REGION Network 3: Дискретные входы состояния НБ
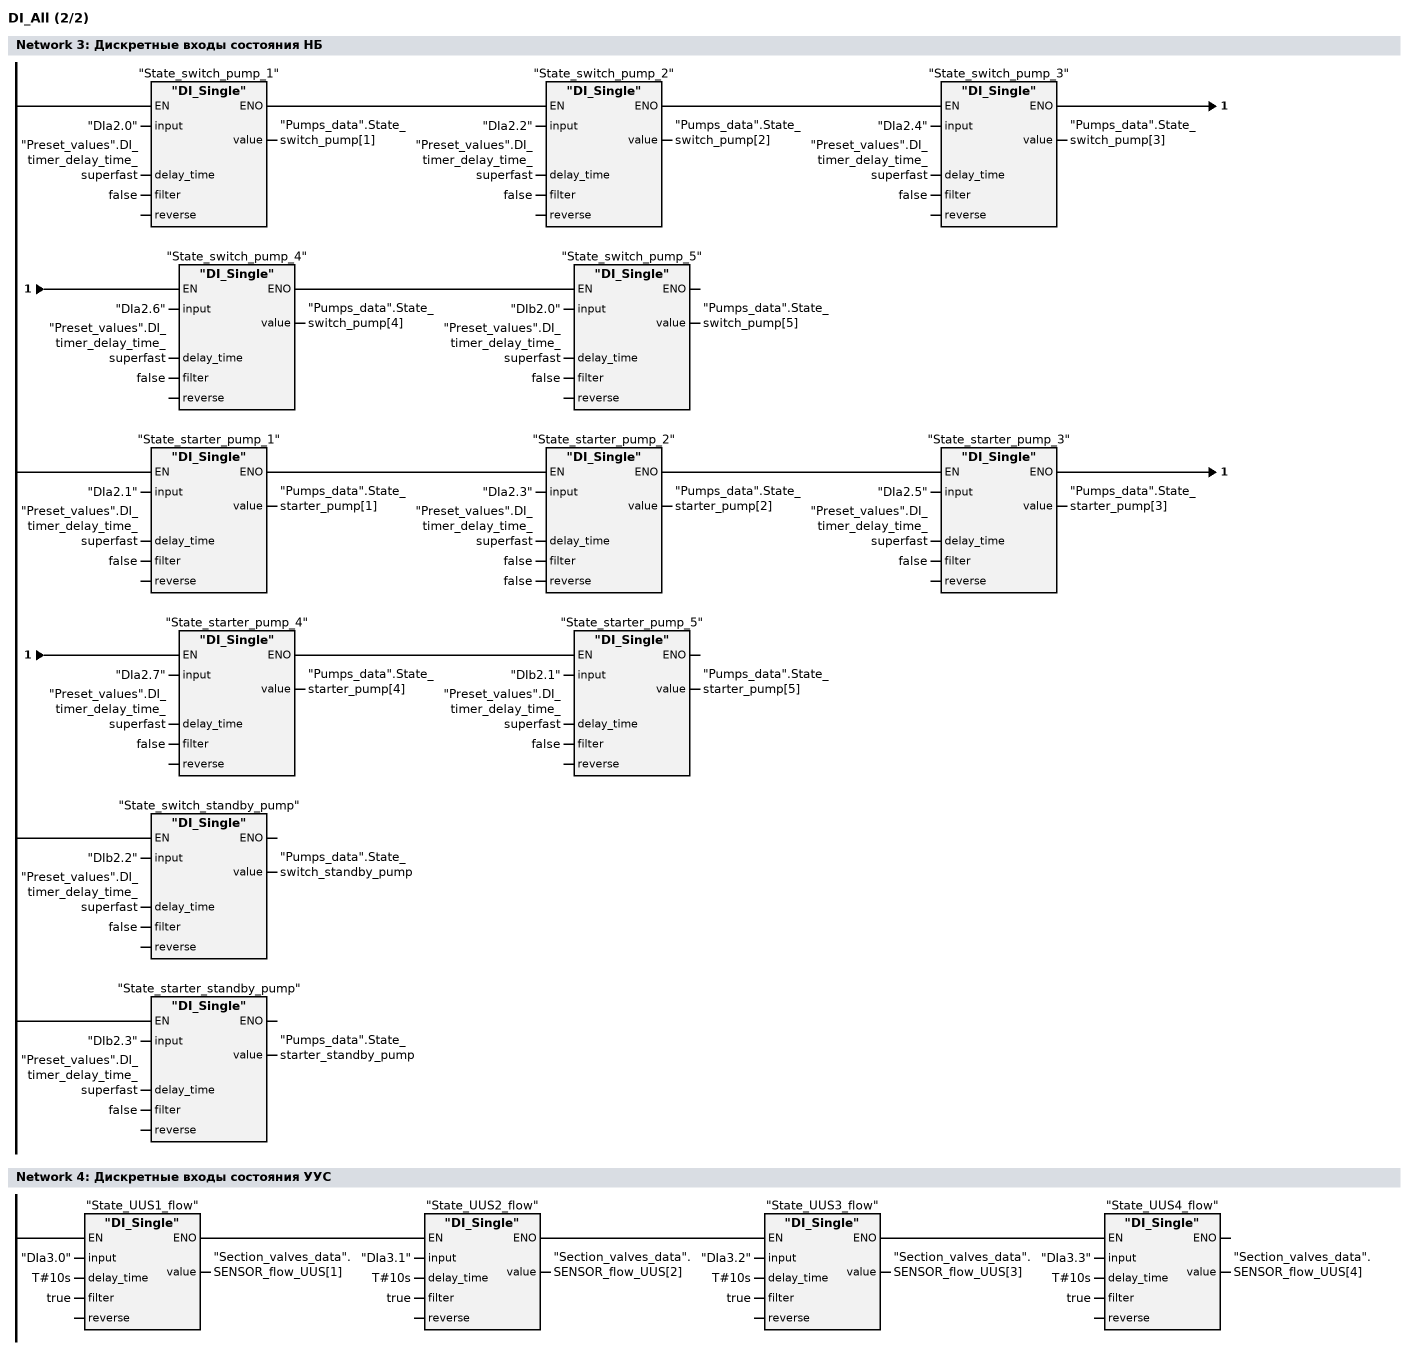
   RUNG wire#powerrail
      "State_switch_pump_1"(input := "DIa2.0", delay_time := "Preset_values".DI_timer_delay_time_superfast, filter := false, reverse :=, value => "Pumps_data".State_switch_pump[1])
      "State_switch_pump_2"(input := "DIa2.2", delay_time := "Preset_values".DI_timer_delay_time_superfast, filter := false, reverse :=, value => "Pumps_data".State_switch_pump[2])
      "State_switch_pump_3"(input := "DIa2.4", delay_time := "Preset_values".DI_timer_delay_time_superfast, filter := false, reverse :=, value => "Pumps_data".State_switch_pump[3])
      "State_switch_pump_4"(input := "DIa2.6", delay_time := "Preset_values".DI_timer_delay_time_superfast, filter := false, reverse :=, value => "Pumps_data".State_switch_pump[4])
      "State_switch_pump_5"(input := "DIb2.0", delay_time := "Preset_values".DI_timer_delay_time_superfast, filter := false, reverse :=, value => "Pumps_data".State_switch_pump[5])
   END_RUNG
   RUNG wire#powerrail
      "State_starter_pump_1"(input := "DIa2.1", delay_time := "Preset_values".DI_timer_delay_time_superfast, filter := false, reverse :=, value => "Pumps_data".State_starter_pump[1])
      "State_starter_pump_2"(input := "DIa2.3", delay_time := "Preset_values".DI_timer_delay_time_superfast, filter := false, reverse := false, value => "Pumps_data".State_starter_pump[2])
      "State_starter_pump_3"(input := "DIa2.5", delay_time := "Preset_values".DI_timer_delay_time_superfast, filter := false, reverse :=, value => "Pumps_data".State_starter_pump[3])
      "State_starter_pump_4"(input := "DIa2.7", delay_time := "Preset_values".DI_timer_delay_time_superfast, filter := false, reverse :=, value => "Pumps_data".State_starter_pump[4])
      "State_starter_pump_5"(input := "DIb2.1", delay_time := "Preset_values".DI_timer_delay_time_superfast, filter := false, reverse :=, value => "Pumps_data".State_starter_pump[5])
   END_RUNG
   RUNG wire#powerrail
      "State_switch_standby_pump"(input := "DIb2.2", delay_time := "Preset_values".DI_timer_delay_time_superfast, filter := false, reverse :=, value => "Pumps_data".State_switch_standby_pump)
   END_RUNG
   RUNG wire#powerrail
      "State_starter_standby_pump"(input := "DIb2.3", delay_time := "Preset_values".DI_timer_delay_time_superfast, filter := false, reverse :=, value => "Pumps_data".State_starter_standby_pump)
   END_RUNG
   // the same network as SCL:
   "State_switch_pump_1"(input := "DIa2.0",   // "DI_Single"
                         delay_time := "Preset_values".DI_timer_delay_time_superfast,
                         filter := false,
                         value => "Pumps_data".State_switch_pump[1],
                         ENO => #_w1);
   "State_switch_pump_2"(EN := #_w1,   // "DI_Single"
                         input := "DIa2.2",
                         delay_time := "Preset_values".DI_timer_delay_time_superfast,
                         filter := false,
                         value => "Pumps_data".State_switch_pump[2],
                         ENO => #_w2);
   "State_switch_pump_3"(EN := #_w2,   // "DI_Single"
                         input := "DIa2.4",
                         delay_time := "Preset_values".DI_timer_delay_time_superfast,
                         filter := false,
                         value => "Pumps_data".State_switch_pump[3],
                         ENO => #_w3);
   "State_switch_pump_4"(EN := #_w3,   // "DI_Single"
                         input := "DIa2.6",
                         delay_time := "Preset_values".DI_timer_delay_time_superfast,
                         filter := false,
                         value => "Pumps_data".State_switch_pump[4],
                         ENO => #_w4);
   IF #_w4 THEN
       "State_switch_pump_5"(input := "DIb2.0",   // "DI_Single"
                             delay_time := "Preset_values".DI_timer_delay_time_superfast,
                             filter := false,
                             value => "Pumps_data".State_switch_pump[5]);
   END_IF;
   "State_starter_pump_1"(input := "DIa2.1",   // "DI_Single"
                          delay_time := "Preset_values".DI_timer_delay_time_superfast,
                          filter := false,
                          value => "Pumps_data".State_starter_pump[1],
                          ENO => #_w5);
   "State_starter_pump_2"(EN := #_w5,   // "DI_Single"
                          input := "DIa2.3",
                          delay_time := "Preset_values".DI_timer_delay_time_superfast,
                          filter := false,
                          reverse := false,
                          value => "Pumps_data".State_starter_pump[2],
                          ENO => #_w6);
   "State_starter_pump_3"(EN := #_w6,   // "DI_Single"
                          input := "DIa2.5",
                          delay_time := "Preset_values".DI_timer_delay_time_superfast,
                          filter := false,
                          value => "Pumps_data".State_starter_pump[3],
                          ENO => #_w7);
   "State_starter_pump_4"(EN := #_w7,   // "DI_Single"
                          input := "DIa2.7",
                          delay_time := "Preset_values".DI_timer_delay_time_superfast,
                          filter := false,
                          value => "Pumps_data".State_starter_pump[4],
                          ENO => #_w8);
   IF #_w8 THEN
       "State_starter_pump_5"(input := "DIb2.1",   // "DI_Single"
                              delay_time := "Preset_values".DI_timer_delay_time_superfast,
                              filter := false,
                              value => "Pumps_data".State_starter_pump[5]);
   END_IF;
   "State_switch_standby_pump"(input := "DIb2.2",   // "DI_Single"
                           delay_time := "Preset_values".DI_timer_delay_time_superfast,
                           filter := false,
                           value => "Pumps_data".State_switch_standby_pump);
   "State_starter_standby_pump"(input := "DIb2.3",   // "DI_Single"
                           delay_time := "Preset_values".DI_timer_delay_time_superfast,
                           filter := false,
                           value => "Pumps_data".State_starter_standby_pump);
END_REGION

REGION Network 4: Дискретные входы состояния УУС
   RUNG wire#powerrail
      "State_UUS1_flow"(input := "DIa3.0", delay_time := T#10s, filter := true, reverse :=, value => "Section_valves_data".SENSOR_flow_UUS[1])
      "State_UUS2_flow"(input := "DIa3.1", delay_time := T#10s, filter := true, reverse :=, value => "Section_valves_data".SENSOR_flow_UUS[2])
      "State_UUS3_flow"(input := "DIa3.2", delay_time := T#10s, filter := true, reverse :=, value => "Section_valves_data".SENSOR_flow_UUS[3])
      "State_UUS4_flow"(input := "DIa3.3", delay_time := T#10s, filter := true, reverse :=, value => "Section_valves_data".SENSOR_flow_UUS[4])
   END_RUNG
   // the same network as SCL:
   "State_UUS1_flow"(input := "DIa3.0",   // "DI_Single"
                     delay_time := T#10s,
                     filter := true,
                     value => "Section_valves_data".SENSOR_flow_UUS[1],
                     ENO => #_w1);
   "State_UUS2_flow"(EN := #_w1,   // "DI_Single"
                     input := "DIa3.1",
                     delay_time := T#10s,
                     filter := true,
                     value => "Section_valves_data".SENSOR_flow_UUS[2],
                     ENO => #_w2);
   "State_UUS3_flow"(EN := #_w2,   // "DI_Single"
                     input := "DIa3.2",
                     delay_time := T#10s,
                     filter := true,
                     value => "Section_valves_data".SENSOR_flow_UUS[3],
                     ENO => #_w3);
   IF #_w3 THEN
       "State_UUS4_flow"(input := "DIa3.3",   // "DI_Single"
                         delay_time := T#10s,
                         filter := true,
                         value => "Section_valves_data".SENSOR_flow_UUS[4]);
   END_IF;
END_REGION
END_FUNCTION

FUNCTION "AI_All" : Void   // FC2, LAD
{ S7_Optimized_Access := 'TRUE' }
VERSION : 0.1
   VAR_TEMP   // added for the SCL form of the ladder/FBD networks
      _w1 : Bool;
      _w2 : Bool;
      _w3 : Bool;
      _w4 : Bool;
   END_VAR
BEGIN

REGION Network 1: Аналоговые входы датчиков низкого давления
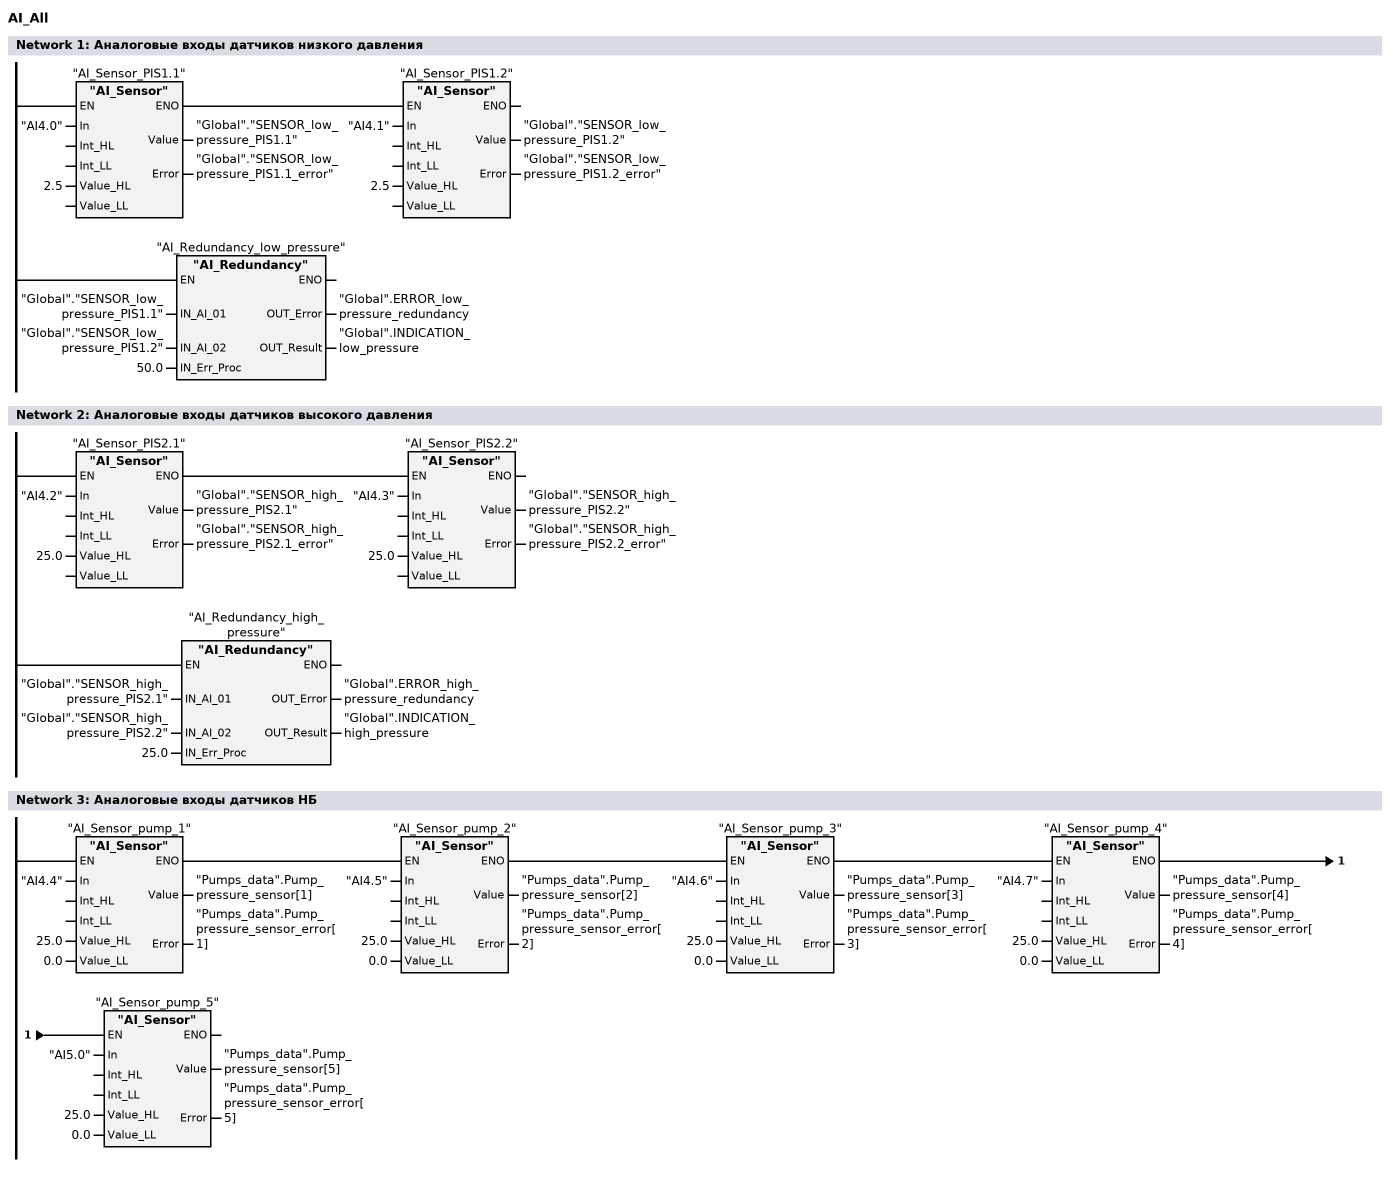
   RUNG wire#powerrail
      "AI_Sensor_PIS1.1"(In := "AI4.0", Int_HL :=, Int_LL :=, Value_HL := 2.5, Value_LL :=, Value => "Global"."SENSOR_low_pressure_PIS1.1", Error => "Global"."SENSOR_low_pressure_PIS1.1_error")
      "AI_Sensor_PIS1.2"(In := "AI4.1", Int_HL :=, Int_LL :=, Value_HL := 2.5, Value_LL :=, Value => "Global"."SENSOR_low_pressure_PIS1.2", Error => "Global"."SENSOR_low_pressure_PIS1.2_error")
   END_RUNG
   RUNG wire#powerrail
      "AI_Redundancy_low_pressure"(IN_AI_01 := "Global"."SENSOR_low_pressure_PIS1.1", IN_AI_02 := "Global"."SENSOR_low_pressure_PIS1.2", IN_Err_Proc := 50.0, OUT_Error => "Global".ERROR_low_pressure_redundancy, OUT_Result => "Global".INDICATION_low_pressure)
   END_RUNG
   // the same network as SCL:
   "AI_Sensor_PIS1.1"(In := "AI4.0",   // "AI_Sensor"
                      Value_HL := 2.5,
                      Value => "Global"."SENSOR_low_pressure_PIS1.1",
                      Error => "Global"."SENSOR_low_pressure_PIS1.1_error",
                      ENO => #_w1);
   IF #_w1 THEN
       "AI_Sensor_PIS1.2"(In := "AI4.1",   // "AI_Sensor"
                          Value_HL := 2.5,
                          Value => "Global"."SENSOR_low_pressure_PIS1.2",
                          Error => "Global"."SENSOR_low_pressure_PIS1.2_error");
   END_IF;
   "AI_Redundancy_low_pressure"(IN_AI_01 := "Global"."SENSOR_low_pressure_PIS1.1",   // "AI_Redundancy"
                           IN_AI_02 := "Global"."SENSOR_low_pressure_PIS1.2",
                           IN_Err_Proc := 50.0,
                           OUT_Error => "Global".ERROR_low_pressure_redundancy,
                           OUT_Result => "Global".INDICATION_low_pressure);
END_REGION

REGION Network 2: Аналоговые входы датчиков высокого давления
   RUNG wire#powerrail
      "AI_Sensor_PIS2.1"(In := "AI4.2", Int_HL :=, Int_LL :=, Value_HL := 25.0, Value_LL :=, Value => "Global"."SENSOR_high_pressure_PIS2.1", Error => "Global"."SENSOR_high_pressure_PIS2.1_error")
      "AI_Sensor_PIS2.2"(In := "AI4.3", Int_HL :=, Int_LL :=, Value_HL := 25.0, Value_LL :=, Value => "Global"."SENSOR_high_pressure_PIS2.2", Error => "Global"."SENSOR_high_pressure_PIS2.2_error")
   END_RUNG
   RUNG wire#powerrail
      "AI_Redundancy_high_pressure"(IN_AI_01 := "Global"."SENSOR_high_pressure_PIS2.1", IN_AI_02 := "Global"."SENSOR_high_pressure_PIS2.2", IN_Err_Proc := 25.0, OUT_Error => "Global".ERROR_high_pressure_redundancy, OUT_Result => "Global".INDICATION_high_pressure)
   END_RUNG
   // the same network as SCL:
   "AI_Sensor_PIS2.1"(In := "AI4.2",   // "AI_Sensor"
                      Value_HL := 25.0,
                      Value => "Global"."SENSOR_high_pressure_PIS2.1",
                      Error => "Global"."SENSOR_high_pressure_PIS2.1_error",
                      ENO => #_w1);
   IF #_w1 THEN
       "AI_Sensor_PIS2.2"(In := "AI4.3",   // "AI_Sensor"
                          Value_HL := 25.0,
                          Value => "Global"."SENSOR_high_pressure_PIS2.2",
                          Error => "Global"."SENSOR_high_pressure_PIS2.2_error");
   END_IF;
   "AI_Redundancy_high_pressure"(IN_AI_01 := "Global"."SENSOR_high_pressure_PIS2.1",   // "AI_Redundancy"
                           IN_AI_02 := "Global"."SENSOR_high_pressure_PIS2.2",
                           IN_Err_Proc := 25.0,
                           OUT_Error => "Global".ERROR_high_pressure_redundancy,
                           OUT_Result => "Global".INDICATION_high_pressure);
END_REGION

REGION Network 3: Аналоговые входы датчиков НБ
   RUNG wire#powerrail
      "AI_Sensor_pump_1"(In := "AI4.4", Int_HL :=, Int_LL :=, Value_HL := 25.0, Value_LL := 0.0, Value => "Pumps_data".Pump_pressure_sensor[1], Error => "Pumps_data".Pump_pressure_sensor_error[1])
      "AI_Sensor_pump_2"(In := "AI4.5", Int_HL :=, Int_LL :=, Value_HL := 25.0, Value_LL := 0.0, Value => "Pumps_data".Pump_pressure_sensor[2], Error => "Pumps_data".Pump_pressure_sensor_error[2])
      "AI_Sensor_pump_3"(In := "AI4.6", Int_HL :=, Int_LL :=, Value_HL := 25.0, Value_LL := 0.0, Value => "Pumps_data".Pump_pressure_sensor[3], Error => "Pumps_data".Pump_pressure_sensor_error[3])
      "AI_Sensor_pump_4"(In := "AI4.7", Int_HL :=, Int_LL :=, Value_HL := 25.0, Value_LL := 0.0, Value => "Pumps_data".Pump_pressure_sensor[4], Error => "Pumps_data".Pump_pressure_sensor_error[4])
      "AI_Sensor_pump_5"(In := "AI5.0", Int_HL :=, Int_LL :=, Value_HL := 25.0, Value_LL := 0.0, Value => "Pumps_data".Pump_pressure_sensor[5], Error => "Pumps_data".Pump_pressure_sensor_error[5])
   END_RUNG
   // the same network as SCL:
   "AI_Sensor_pump_1"(In := "AI4.4",   // "AI_Sensor"
                      Value_HL := 25.0,
                      Value_LL := 0.0,
                      Value => "Pumps_data".Pump_pressure_sensor[1],
                      Error => "Pumps_data".Pump_pressure_sensor_error[1],
                      ENO => #_w1);
   "AI_Sensor_pump_2"(EN := #_w1,   // "AI_Sensor"
                      In := "AI4.5",
                      Value_HL := 25.0,
                      Value_LL := 0.0,
                      Value => "Pumps_data".Pump_pressure_sensor[2],
                      Error => "Pumps_data".Pump_pressure_sensor_error[2],
                      ENO => #_w2);
   "AI_Sensor_pump_3"(EN := #_w2,   // "AI_Sensor"
                      In := "AI4.6",
                      Value_HL := 25.0,
                      Value_LL := 0.0,
                      Value => "Pumps_data".Pump_pressure_sensor[3],
                      Error => "Pumps_data".Pump_pressure_sensor_error[3],
                      ENO => #_w3);
   "AI_Sensor_pump_4"(EN := #_w3,   // "AI_Sensor"
                      In := "AI4.7",
                      Value_HL := 25.0,
                      Value_LL := 0.0,
                      Value => "Pumps_data".Pump_pressure_sensor[4],
                      Error => "Pumps_data".Pump_pressure_sensor_error[4],
                      ENO => #_w4);
   IF #_w4 THEN
       "AI_Sensor_pump_5"(In := "AI5.0",   // "AI_Sensor"
                          Value_HL := 25.0,
                          Value_LL := 0.0,
                          Value => "Pumps_data".Pump_pressure_sensor[5],
                          Error => "Pumps_data".Pump_pressure_sensor_error[5]);
   END_IF;
END_REGION
END_FUNCTION

ORGANIZATION_BLOCK "Main"   // OB1, LAD, ProgramCycle
TITLE = "Main Program Sweep (Cycle)"
{ S7_Optimized_Access := 'TRUE' }
VERSION : 0.1
   VAR_INPUT
      Initial_Call : Bool;   // Initial call of this OB
      Remanence : Bool;   // =True, if remanent data are available
   END_VAR
BEGIN

REGION Network 1: Обработка дискретных и аналоговых сигналов
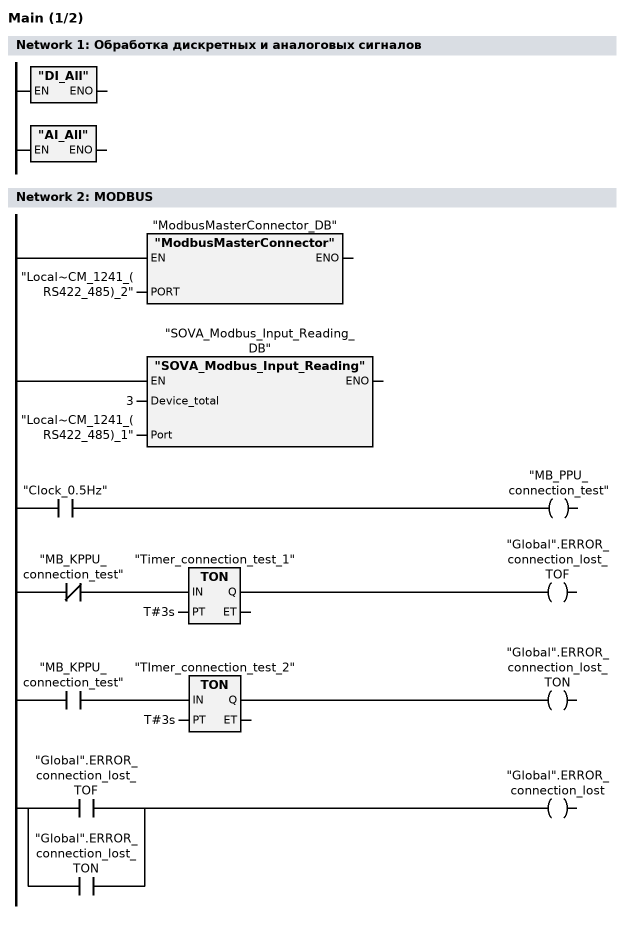
   RUNG wire#powerrail
      "DI_All"()
   END_RUNG
   RUNG wire#powerrail
      "AI_All"()
   END_RUNG
   // the same network as SCL:
   "DI_All"();
   "AI_All"();
END_REGION

REGION Network 2: MODBUS
   "ModbusMasterConnector_DB"(PORT := "Local~CM_1241_(RS422_485)_2");   // "ModbusMasterConnector"
   "SOVA_Modbus_Input_Reading_DB"(Device_total := 3, Port := "Local~CM_1241_(RS422_485)_1");   // "SOVA_Modbus_Input_Reading"
   "MB_PPU_connection_test" := "Clock_0.5Hz";
   "Timer_connection_test_1".TON(IN := NOT "MB_KPPU_connection_test", PT := T#3s);
   "Global".ERROR_connection_lost_TOF := "Timer_connection_test_1".Q;
   "TImer_connection_test_2".TON(IN := "MB_KPPU_connection_test", PT := T#3s);
   "Global".ERROR_connection_lost_TON := "TImer_connection_test_2".Q;
   "Global".ERROR_connection_lost := "Global".ERROR_connection_lost_TOF OR "Global".ERROR_connection_lost_TON;
END_REGION

REGION Network 3: Состояние режима работы ППУ
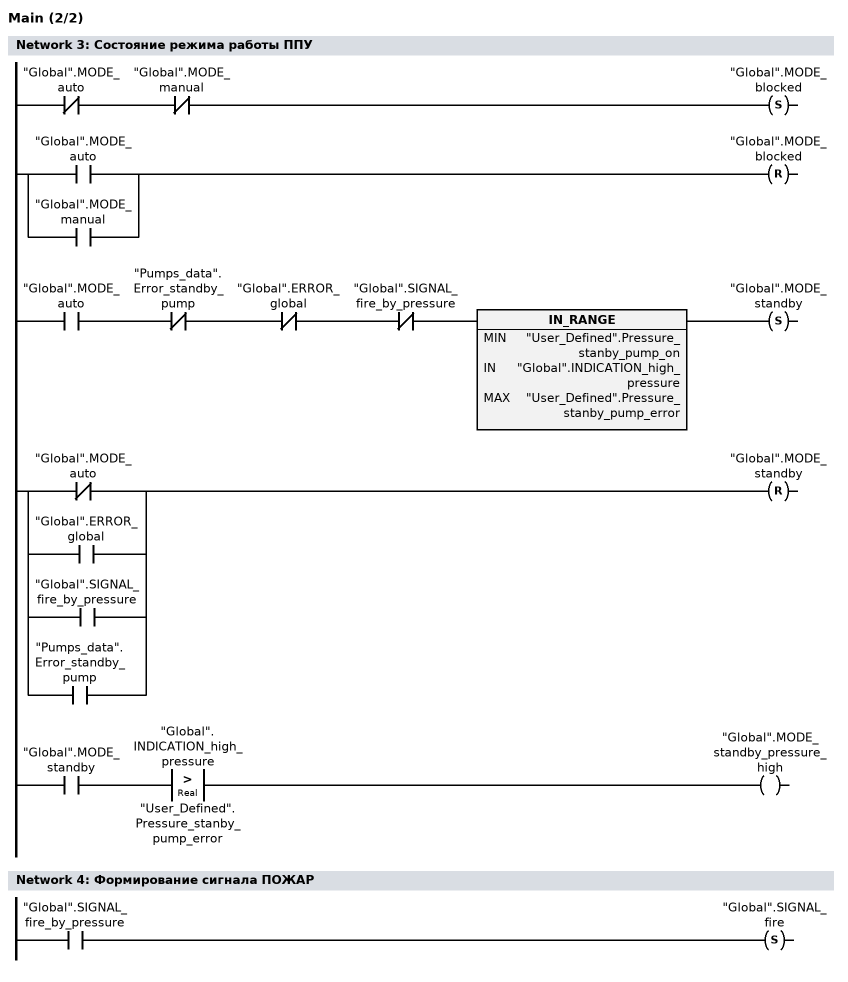
   RUNG wire#powerrail
      I_Contact( "Global".MODE_auto )
      I_Contact( "Global".MODE_manual )
      S_Coil( "Global".MODE_blocked )
   END_RUNG
   RUNG wire#powerrail
      Contact( "Global".MODE_auto )
      wire#w1
      R_Coil( "Global".MODE_blocked )
   END_RUNG
   RUNG wire#powerrail
      Contact( "Global".MODE_manual )
   END_RUNG wire#w1
   RUNG wire#powerrail
      Contact( "Global".MODE_auto )
      I_Contact( "Pumps_data".Error_standby_pump )
      I_Contact( "Global".ERROR_global )
      I_Contact( "Global".SIGNAL_fire_by_pressure )
      { S7_Templates := "SrcType := Real" } InRange(min := "User_Defined".Pressure_stanby_pump_on, in := "Global".INDICATION_high_pressure, max := "User_Defined".Pressure_stanby_pump_error)
      S_Coil( "Global".MODE_standby )
   END_RUNG
   RUNG wire#powerrail
      I_Contact( "Global".MODE_auto )
      wire#w2
      R_Coil( "Global".MODE_standby )
   END_RUNG
   RUNG wire#powerrail
      Contact( "Global".ERROR_global )
   END_RUNG wire#w2
   RUNG wire#powerrail
      Contact( "Global".SIGNAL_fire_by_pressure )
   END_RUNG wire#w2
   RUNG wire#powerrail
      Contact( "Pumps_data".Error_standby_pump )
   END_RUNG wire#w2
   RUNG wire#powerrail
      Contact( "Global".MODE_standby )
      { S7_Templates := "SrcType := Real" } GT_Contact(in1 := "Global".INDICATION_high_pressure, in2 := "User_Defined".Pressure_stanby_pump_error)
      Coil( "Global".MODE_standby_pressure_high )
   END_RUNG
   // the same network as SCL:
   IF NOT "Global".MODE_auto AND NOT "Global".MODE_manual THEN "Global".MODE_blocked := TRUE; END_IF;
   IF "Global".MODE_auto OR "Global".MODE_manual THEN "Global".MODE_blocked := FALSE; END_IF;
   IF "Global".MODE_auto AND NOT "Pumps_data".Error_standby_pump AND NOT "Global".ERROR_global AND NOT "Global".SIGNAL_fire_by_pressure AND ("User_Defined".Pressure_stanby_pump_on <= "Global".INDICATION_high_pressure) AND ("Global".INDICATION_high_pressure <= "User_Defined".Pressure_stanby_pump_error) THEN
       "Global".MODE_standby := TRUE;
   END_IF;
   IF NOT "Global".MODE_auto OR "Global".ERROR_global OR "Global".SIGNAL_fire_by_pressure OR "Pumps_data".Error_standby_pump THEN
       "Global".MODE_standby := FALSE;
   END_IF;
   "Global".MODE_standby_pressure_high := "Global".MODE_standby AND ("Global".INDICATION_high_pressure > "User_Defined".Pressure_stanby_pump_error);
END_REGION

REGION Network 4: Формирование сигнала ПОЖАР
   RUNG wire#powerrail
      Contact( "Global".SIGNAL_fire_by_pressure )
      S_Coil( "Global".SIGNAL_fire )
   END_RUNG
   // the same network as SCL:
   IF "Global".SIGNAL_fire_by_pressure THEN "Global".SIGNAL_fire := TRUE; END_IF;
END_REGION

REGION Network 5 (SCL): Pump Work Counter
   IF "Pumps_data".State_work_pump[1] THEN
       "Pumps_data".Pump_work_counter_arr[1] := 1;
   ELSE
       "Pumps_data".Pump_work_counter_arr[1] := 0;
   END_IF;

   IF "Pumps_data".State_work_pump[2] THEN
       "Pumps_data".Pump_work_counter_arr[2] := 1;
   ELSE
       "Pumps_data".Pump_work_counter_arr[2] := 0;
   END_IF;

   IF "Pumps_data".State_work_pump[3] THEN
       "Pumps_data".Pump_work_counter_arr[3] := 1;
   ELSE
       "Pumps_data".Pump_work_counter_arr[3] := 0;
   END_IF;

   IF "Pumps_data".State_work_pump[4] THEN
       "Pumps_data".Pump_work_counter_arr[4] := 1;
   ELSE
       "Pumps_data".Pump_work_counter_arr[4] := 0;
   END_IF;

   IF "Pumps_data".State_work_pump[5] THEN
       "Pumps_data".Pump_work_counter_arr[5] := 1;
   ELSE
       "Pumps_data".Pump_work_counter_arr[5] := 0;
   END_IF;

   IF "Pumps_data".State_work_pump[6] THEN
       "Pumps_data".Pump_work_counter_arr[6] := 1;
   ELSE
       "Pumps_data".Pump_work_counter_arr[6] := 0;
   END_IF;

   IF "Pumps_data".State_work_pump[7] THEN
       "Pumps_data".Pump_work_counter_arr[7] := 1;
   ELSE
       "Pumps_data".Pump_work_counter_arr[7] := 0;
   END_IF;

   IF "Pumps_data".State_work_pump[8] THEN
       "Pumps_data".Pump_work_counter_arr[8] := 1;
   ELSE
       "Pumps_data".Pump_work_counter_arr[8] := 0;
   END_IF;

   IF "Pumps_data".State_work_pump[9] THEN
       "Pumps_data".Pump_work_counter_arr[9] := 1;
   ELSE
       "Pumps_data".Pump_work_counter_arr[9] := 0;
   END_IF;

   IF "Pumps_data".State_work_pump[10] THEN
       "Pumps_data".Pump_work_counter_arr[10] := 1;
   ELSE
       "Pumps_data".Pump_work_counter_arr[10] := 0;
   END_IF;

   "Pumps_data".pump_work_counter := "Pumps_data".Pump_work_counter_arr[1] +
   "Pumps_data".Pump_work_counter_arr[2] + "Pumps_data".Pump_work_counter_arr[3] +
   "Pumps_data".Pump_work_counter_arr[4] + "Pumps_data".Pump_work_counter_arr[5] +
   "Pumps_data".Pump_work_counter_arr[6] + "Pumps_data".Pump_work_counter_arr[7] +
   "Pumps_data".Pump_work_counter_arr[8] + "Pumps_data".Pump_work_counter_arr[9] +
   "Pumps_data".Pump_work_counter_arr[10];
END_REGION
END_ORGANIZATION_BLOCK

ORGANIZATION_BLOCK "Errors"   // OB123, LAD, ProgramCycle
TITLE = "Main Program Sweep (Cycle)"
{ S7_Optimized_Access := 'TRUE' }
VERSION : 0.1
   VAR_INPUT
      Initial_Call : Bool;   // Initial call of this OB
      Remanence : Bool;   // =True, if remanent data are available
   END_VAR
   VAR_TEMP   // added for the SCL form of the ladder/FBD networks
      _w1 : Bool;
      _w2 : Bool;
      _w3 : Bool;
      _w4 : Bool;
      _w5 : Bool;
      _w6 : Bool;
      _w7 : Bool;
      _w8 : Bool;
   END_VAR
BEGIN

REGION Network 1: Недостаточное входное давление
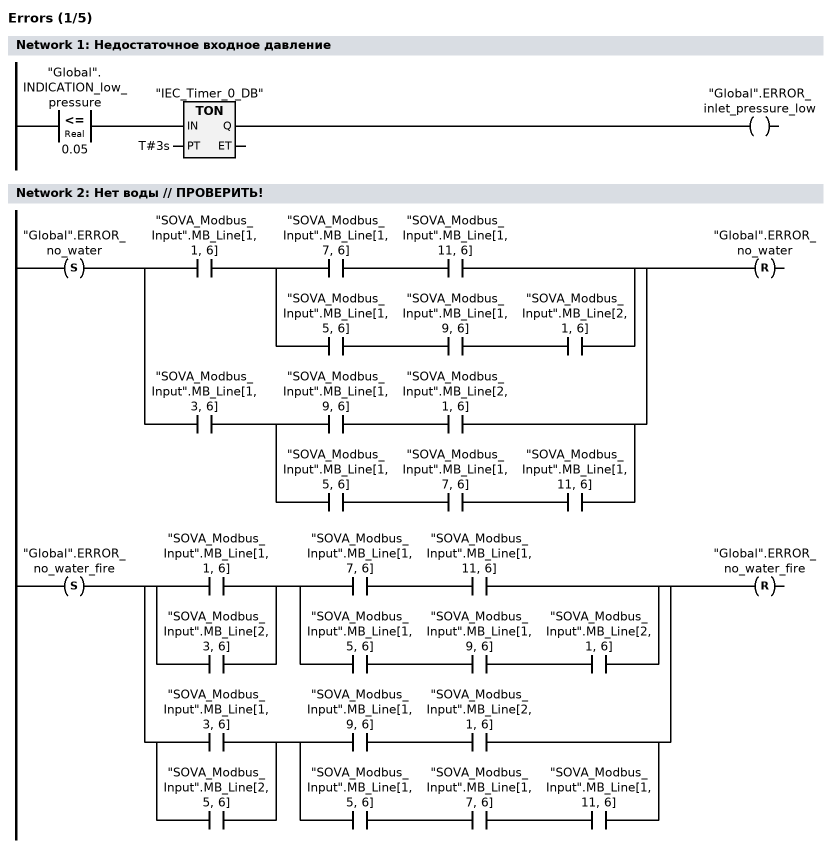
   "IEC_Timer_0_DB".TON(IN := "Global".INDICATION_low_pressure <= 0.05, PT := T#3s);
   "Global".ERROR_inlet_pressure_low := "IEC_Timer_0_DB".Q;
END_REGION

REGION Network 2: Нет воды // ПРОВЕРИТЬ!
   RUNG wire#powerrail
      S_Coil( "Global".ERROR_no_water )
      wire#w1
      Contact( "SOVA_Modbus_Input".MB_Line[1, 1, 6] )
      wire#w2
      Contact( "SOVA_Modbus_Input".MB_Line[1, 7, 6] )
      Contact( "SOVA_Modbus_Input".MB_Line[1, 11, 6] )
      wire#w3
      R_Coil( "Global".ERROR_no_water )
   END_RUNG
   RUNG wire#w2
      Contact( "SOVA_Modbus_Input".MB_Line[1, 5, 6] )
      Contact( "SOVA_Modbus_Input".MB_Line[1, 9, 6] )
      Contact( "SOVA_Modbus_Input".MB_Line[2, 1, 6] )
   END_RUNG wire#w3
   RUNG wire#w1
      Contact( "SOVA_Modbus_Input".MB_Line[1, 3, 6] )
      wire#w4
      Contact( "SOVA_Modbus_Input".MB_Line[1, 9, 6] )
      Contact( "SOVA_Modbus_Input".MB_Line[2, 1, 6] )
   END_RUNG wire#w3
   RUNG wire#w4
      Contact( "SOVA_Modbus_Input".MB_Line[1, 5, 6] )
      Contact( "SOVA_Modbus_Input".MB_Line[1, 7, 6] )
      Contact( "SOVA_Modbus_Input".MB_Line[1, 11, 6] )
   END_RUNG wire#w3
   RUNG wire#powerrail
      S_Coil( "Global".ERROR_no_water_fire )
      wire#w5
      Contact( "SOVA_Modbus_Input".MB_Line[1, 1, 6] )
      wire#w6
      Contact( "SOVA_Modbus_Input".MB_Line[1, 7, 6] )
      Contact( "SOVA_Modbus_Input".MB_Line[1, 11, 6] )
      wire#w7
      R_Coil( "Global".ERROR_no_water_fire )
   END_RUNG
   RUNG wire#w5
      Contact( "SOVA_Modbus_Input".MB_Line[2, 3, 6] )
   END_RUNG wire#w6
   RUNG wire#w6
      Contact( "SOVA_Modbus_Input".MB_Line[1, 5, 6] )
      Contact( "SOVA_Modbus_Input".MB_Line[1, 9, 6] )
      Contact( "SOVA_Modbus_Input".MB_Line[2, 1, 6] )
   END_RUNG wire#w7
   RUNG wire#w5
      Contact( "SOVA_Modbus_Input".MB_Line[1, 3, 6] )
      wire#w8
      Contact( "SOVA_Modbus_Input".MB_Line[1, 9, 6] )
      Contact( "SOVA_Modbus_Input".MB_Line[2, 1, 6] )
   END_RUNG wire#w7
   RUNG wire#w5
      Contact( "SOVA_Modbus_Input".MB_Line[2, 5, 6] )
   END_RUNG wire#w8
   RUNG wire#w8
      Contact( "SOVA_Modbus_Input".MB_Line[1, 5, 6] )
      Contact( "SOVA_Modbus_Input".MB_Line[1, 7, 6] )
      Contact( "SOVA_Modbus_Input".MB_Line[1, 11, 6] )
   END_RUNG wire#w7
   // the same network as SCL:
   "Global".ERROR_no_water := TRUE;
   IF ("SOVA_Modbus_Input".MB_Line[1, 1, 6] AND (("SOVA_Modbus_Input".MB_Line[1, 7, 6] AND "SOVA_Modbus_Input".MB_Line[1, 11, 6]) OR ("SOVA_Modbus_Input".MB_Line[1, 5, 6] AND "SOVA_Modbus_Input".MB_Line[1, 9, 6] AND "SOVA_Modbus_Input".MB_Line[2, 1, 6]))) OR ("SOVA_Modbus_Input".MB_Line[1, 3, 6] AND (("SOVA_Modbus_Input".MB_Line[1, 9, 6] AND "SOVA_Modbus_Input".MB_Line[2, 1, 6]) OR ("SOVA_Modbus_Input".MB_Line[1, 5, 6] AND "SOVA_Modbus_Input".MB_Line[1, 7, 6] AND "SOVA_Modbus_Input".MB_Line[1, 11, 6]))) THEN
       "Global".ERROR_no_water := FALSE;
   END_IF;
   "Global".ERROR_no_water_fire := TRUE;
   IF (("SOVA_Modbus_Input".MB_Line[1, 1, 6] OR "SOVA_Modbus_Input".MB_Line[2, 3, 6]) AND (("SOVA_Modbus_Input".MB_Line[1, 7, 6] AND "SOVA_Modbus_Input".MB_Line[1, 11, 6]) OR ("SOVA_Modbus_Input".MB_Line[1, 5, 6] AND "SOVA_Modbus_Input".MB_Line[1, 9, 6] AND "SOVA_Modbus_Input".MB_Line[2, 1, 6]))) OR (("SOVA_Modbus_Input".MB_Line[1, 3, 6] OR "SOVA_Modbus_Input".MB_Line[2, 5, 6]) AND (("SOVA_Modbus_Input".MB_Line[1, 9, 6] AND "SOVA_Modbus_Input".MB_Line[2, 1, 6]) OR ("SOVA_Modbus_Input".MB_Line[1, 5, 6] AND "SOVA_Modbus_Input".MB_Line[1, 7, 6] AND "SOVA_Modbus_Input".MB_Line[1, 11, 6]))) THEN
       "Global".ERROR_no_water_fire := FALSE;
   END_IF;
END_REGION

REGION Network 3: Неисправность вводных задвижек
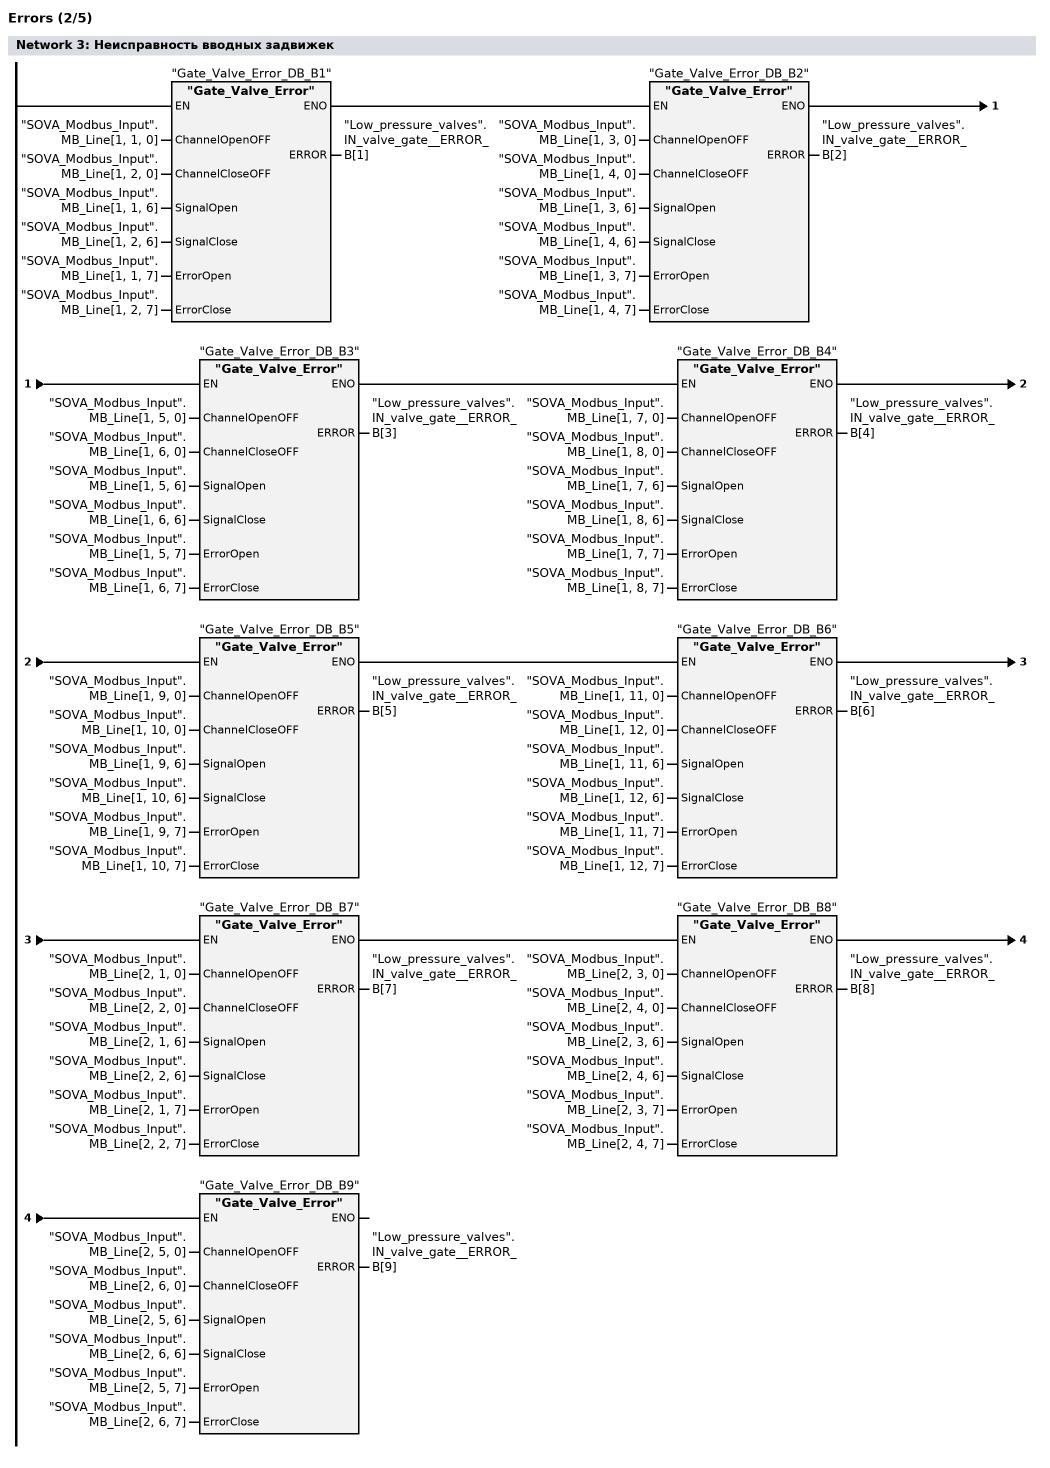
   RUNG wire#powerrail
      "Gate_Valve_Error_DB_B1"(ChannelOpenOFF := "SOVA_Modbus_Input".MB_Line[1, 1, 0], ChannelCloseOFF := "SOVA_Modbus_Input".MB_Line[1, 2, 0], SignalOpen := "SOVA_Modbus_Input".MB_Line[1, 1, 6], SignalClose := "SOVA_Modbus_Input".MB_Line[1, 2, 6], ErrorOpen := "SOVA_Modbus_Input".MB_Line[1, 1, 7], ErrorClose := "SOVA_Modbus_Input".MB_Line[1, 2, 7], ERROR => "Low_pressure_valves".IN_valve_gate__ERROR_B[1])
      "Gate_Valve_Error_DB_B2"(ChannelOpenOFF := "SOVA_Modbus_Input".MB_Line[1, 3, 0], ChannelCloseOFF := "SOVA_Modbus_Input".MB_Line[1, 4, 0], SignalOpen := "SOVA_Modbus_Input".MB_Line[1, 3, 6], SignalClose := "SOVA_Modbus_Input".MB_Line[1, 4, 6], ErrorOpen := "SOVA_Modbus_Input".MB_Line[1, 3, 7], ErrorClose := "SOVA_Modbus_Input".MB_Line[1, 4, 7], ERROR => "Low_pressure_valves".IN_valve_gate__ERROR_B[2])
      "Gate_Valve_Error_DB_B3"(ChannelOpenOFF := "SOVA_Modbus_Input".MB_Line[1, 5, 0], ChannelCloseOFF := "SOVA_Modbus_Input".MB_Line[1, 6, 0], SignalOpen := "SOVA_Modbus_Input".MB_Line[1, 5, 6], SignalClose := "SOVA_Modbus_Input".MB_Line[1, 6, 6], ErrorOpen := "SOVA_Modbus_Input".MB_Line[1, 5, 7], ErrorClose := "SOVA_Modbus_Input".MB_Line[1, 6, 7], ERROR => "Low_pressure_valves".IN_valve_gate__ERROR_B[3])
      "Gate_Valve_Error_DB_B4"(ChannelOpenOFF := "SOVA_Modbus_Input".MB_Line[1, 7, 0], ChannelCloseOFF := "SOVA_Modbus_Input".MB_Line[1, 8, 0], SignalOpen := "SOVA_Modbus_Input".MB_Line[1, 7, 6], SignalClose := "SOVA_Modbus_Input".MB_Line[1, 8, 6], ErrorOpen := "SOVA_Modbus_Input".MB_Line[1, 7, 7], ErrorClose := "SOVA_Modbus_Input".MB_Line[1, 8, 7], ERROR => "Low_pressure_valves".IN_valve_gate__ERROR_B[4])
      "Gate_Valve_Error_DB_B5"(ChannelOpenOFF := "SOVA_Modbus_Input".MB_Line[1, 9, 0], ChannelCloseOFF := "SOVA_Modbus_Input".MB_Line[1, 10, 0], SignalOpen := "SOVA_Modbus_Input".MB_Line[1, 9, 6], SignalClose := "SOVA_Modbus_Input".MB_Line[1, 10, 6], ErrorOpen := "SOVA_Modbus_Input".MB_Line[1, 9, 7], ErrorClose := "SOVA_Modbus_Input".MB_Line[1, 10, 7], ERROR => "Low_pressure_valves".IN_valve_gate__ERROR_B[5])
      "Gate_Valve_Error_DB_B6"(ChannelOpenOFF := "SOVA_Modbus_Input".MB_Line[1, 11, 0], ChannelCloseOFF := "SOVA_Modbus_Input".MB_Line[1, 12, 0], SignalOpen := "SOVA_Modbus_Input".MB_Line[1, 11, 6], SignalClose := "SOVA_Modbus_Input".MB_Line[1, 12, 6], ErrorOpen := "SOVA_Modbus_Input".MB_Line[1, 11, 7], ErrorClose := "SOVA_Modbus_Input".MB_Line[1, 12, 7], ERROR => "Low_pressure_valves".IN_valve_gate__ERROR_B[6])
      "Gate_Valve_Error_DB_B7"(ChannelOpenOFF := "SOVA_Modbus_Input".MB_Line[2, 1, 0], ChannelCloseOFF := "SOVA_Modbus_Input".MB_Line[2, 2, 0], SignalOpen := "SOVA_Modbus_Input".MB_Line[2, 1, 6], SignalClose := "SOVA_Modbus_Input".MB_Line[2, 2, 6], ErrorOpen := "SOVA_Modbus_Input".MB_Line[2, 1, 7], ErrorClose := "SOVA_Modbus_Input".MB_Line[2, 2, 7], ERROR => "Low_pressure_valves".IN_valve_gate__ERROR_B[7])
      "Gate_Valve_Error_DB_B8"(ChannelOpenOFF := "SOVA_Modbus_Input".MB_Line[2, 3, 0], ChannelCloseOFF := "SOVA_Modbus_Input".MB_Line[2, 4, 0], SignalOpen := "SOVA_Modbus_Input".MB_Line[2, 3, 6], SignalClose := "SOVA_Modbus_Input".MB_Line[2, 4, 6], ErrorOpen := "SOVA_Modbus_Input".MB_Line[2, 3, 7], ErrorClose := "SOVA_Modbus_Input".MB_Line[2, 4, 7], ERROR => "Low_pressure_valves".IN_valve_gate__ERROR_B[8])
      "Gate_Valve_Error_DB_B9"(ChannelOpenOFF := "SOVA_Modbus_Input".MB_Line[2, 5, 0], ChannelCloseOFF := "SOVA_Modbus_Input".MB_Line[2, 6, 0], SignalOpen := "SOVA_Modbus_Input".MB_Line[2, 5, 6], SignalClose := "SOVA_Modbus_Input".MB_Line[2, 6, 6], ErrorOpen := "SOVA_Modbus_Input".MB_Line[2, 5, 7], ErrorClose := "SOVA_Modbus_Input".MB_Line[2, 6, 7], ERROR => "Low_pressure_valves".IN_valve_gate__ERROR_B[9])
   END_RUNG
   // the same network as SCL:
   "Gate_Valve_Error_DB_B1"(ChannelOpenOFF := "SOVA_Modbus_Input".MB_Line[1, 1, 0],   // "Gate_Valve_Error"
                           ChannelCloseOFF := "SOVA_Modbus_Input".MB_Line[1, 2, 0],
                           SignalOpen := "SOVA_Modbus_Input".MB_Line[1, 1, 6],
                           SignalClose := "SOVA_Modbus_Input".MB_Line[1, 2, 6],
                           ErrorOpen := "SOVA_Modbus_Input".MB_Line[1, 1, 7],
                           ErrorClose := "SOVA_Modbus_Input".MB_Line[1, 2, 7],
                           ERROR => "Low_pressure_valves".IN_valve_gate__ERROR_B[1],
                           ENO => #_w1);
   "Gate_Valve_Error_DB_B2"(EN := #_w1,   // "Gate_Valve_Error"
                           ChannelOpenOFF := "SOVA_Modbus_Input".MB_Line[1, 3, 0],
                           ChannelCloseOFF := "SOVA_Modbus_Input".MB_Line[1, 4, 0],
                           SignalOpen := "SOVA_Modbus_Input".MB_Line[1, 3, 6],
                           SignalClose := "SOVA_Modbus_Input".MB_Line[1, 4, 6],
                           ErrorOpen := "SOVA_Modbus_Input".MB_Line[1, 3, 7],
                           ErrorClose := "SOVA_Modbus_Input".MB_Line[1, 4, 7],
                           ERROR => "Low_pressure_valves".IN_valve_gate__ERROR_B[2],
                           ENO => #_w2);
   "Gate_Valve_Error_DB_B3"(EN := #_w2,   // "Gate_Valve_Error"
                           ChannelOpenOFF := "SOVA_Modbus_Input".MB_Line[1, 5, 0],
                           ChannelCloseOFF := "SOVA_Modbus_Input".MB_Line[1, 6, 0],
                           SignalOpen := "SOVA_Modbus_Input".MB_Line[1, 5, 6],
                           SignalClose := "SOVA_Modbus_Input".MB_Line[1, 6, 6],
                           ErrorOpen := "SOVA_Modbus_Input".MB_Line[1, 5, 7],
                           ErrorClose := "SOVA_Modbus_Input".MB_Line[1, 6, 7],
                           ERROR => "Low_pressure_valves".IN_valve_gate__ERROR_B[3],
                           ENO => #_w3);
   "Gate_Valve_Error_DB_B4"(EN := #_w3,   // "Gate_Valve_Error"
                           ChannelOpenOFF := "SOVA_Modbus_Input".MB_Line[1, 7, 0],
                           ChannelCloseOFF := "SOVA_Modbus_Input".MB_Line[1, 8, 0],
                           SignalOpen := "SOVA_Modbus_Input".MB_Line[1, 7, 6],
                           SignalClose := "SOVA_Modbus_Input".MB_Line[1, 8, 6],
                           ErrorOpen := "SOVA_Modbus_Input".MB_Line[1, 7, 7],
                           ErrorClose := "SOVA_Modbus_Input".MB_Line[1, 8, 7],
                           ERROR => "Low_pressure_valves".IN_valve_gate__ERROR_B[4],
                           ENO => #_w4);
   "Gate_Valve_Error_DB_B5"(EN := #_w4,   // "Gate_Valve_Error"
                           ChannelOpenOFF := "SOVA_Modbus_Input".MB_Line[1, 9, 0],
                           ChannelCloseOFF := "SOVA_Modbus_Input".MB_Line[1, 10, 0],
                           SignalOpen := "SOVA_Modbus_Input".MB_Line[1, 9, 6],
                           SignalClose := "SOVA_Modbus_Input".MB_Line[1, 10, 6],
                           ErrorOpen := "SOVA_Modbus_Input".MB_Line[1, 9, 7],
                           ErrorClose := "SOVA_Modbus_Input".MB_Line[1, 10, 7],
                           ERROR => "Low_pressure_valves".IN_valve_gate__ERROR_B[5],
                           ENO => #_w5);
   "Gate_Valve_Error_DB_B6"(EN := #_w5,   // "Gate_Valve_Error"
                           ChannelOpenOFF := "SOVA_Modbus_Input".MB_Line[1, 11, 0],
                           ChannelCloseOFF := "SOVA_Modbus_Input".MB_Line[1, 12, 0],
                           SignalOpen := "SOVA_Modbus_Input".MB_Line[1, 11, 6],
                           SignalClose := "SOVA_Modbus_Input".MB_Line[1, 12, 6],
                           ErrorOpen := "SOVA_Modbus_Input".MB_Line[1, 11, 7],
                           ErrorClose := "SOVA_Modbus_Input".MB_Line[1, 12, 7],
                           ERROR => "Low_pressure_valves".IN_valve_gate__ERROR_B[6],
                           ENO => #_w6);
   "Gate_Valve_Error_DB_B7"(EN := #_w6,   // "Gate_Valve_Error"
                           ChannelOpenOFF := "SOVA_Modbus_Input".MB_Line[2, 1, 0],
                           ChannelCloseOFF := "SOVA_Modbus_Input".MB_Line[2, 2, 0],
                           SignalOpen := "SOVA_Modbus_Input".MB_Line[2, 1, 6],
                           SignalClose := "SOVA_Modbus_Input".MB_Line[2, 2, 6],
                           ErrorOpen := "SOVA_Modbus_Input".MB_Line[2, 1, 7],
                           ErrorClose := "SOVA_Modbus_Input".MB_Line[2, 2, 7],
                           ERROR => "Low_pressure_valves".IN_valve_gate__ERROR_B[7],
                           ENO => #_w7);
   "Gate_Valve_Error_DB_B8"(EN := #_w7,   // "Gate_Valve_Error"
                           ChannelOpenOFF := "SOVA_Modbus_Input".MB_Line[2, 3, 0],
                           ChannelCloseOFF := "SOVA_Modbus_Input".MB_Line[2, 4, 0],
                           SignalOpen := "SOVA_Modbus_Input".MB_Line[2, 3, 6],
                           SignalClose := "SOVA_Modbus_Input".MB_Line[2, 4, 6],
                           ErrorOpen := "SOVA_Modbus_Input".MB_Line[2, 3, 7],
                           ErrorClose := "SOVA_Modbus_Input".MB_Line[2, 4, 7],
                           ERROR => "Low_pressure_valves".IN_valve_gate__ERROR_B[8],
                           ENO => #_w8);
   IF #_w8 THEN
       "Gate_Valve_Error_DB_B9"(ChannelOpenOFF := "SOVA_Modbus_Input".MB_Line[2, 5, 0],   // "Gate_Valve_Error"
                               ChannelCloseOFF := "SOVA_Modbus_Input".MB_Line[2, 6, 0],
                               SignalOpen := "SOVA_Modbus_Input".MB_Line[2, 5, 6],
                               SignalClose := "SOVA_Modbus_Input".MB_Line[2, 6, 6],
                               ErrorOpen := "SOVA_Modbus_Input".MB_Line[2, 5, 7],
                               ErrorClose := "SOVA_Modbus_Input".MB_Line[2, 6, 7],
                               ERROR => "Low_pressure_valves".IN_valve_gate__ERROR_B[9]);
   END_IF;
END_REGION

REGION Network 4 (SCL): Неисправность любой вводной задвижки
   IF  "Low_pressure_valves"."IN_valve_gate__ERROR_B"[1] OR
       "Low_pressure_valves"."IN_valve_gate__ERROR_B"[2] OR
       "Low_pressure_valves"."IN_valve_gate__ERROR_B"[3] OR
       "Low_pressure_valves"."IN_valve_gate__ERROR_B"[4] OR
       "Low_pressure_valves"."IN_valve_gate__ERROR_B"[5] OR
       "Low_pressure_valves"."IN_valve_gate__ERROR_B"[6] OR
       "Low_pressure_valves"."IN_valve_gate__ERROR_B"[7] OR
       "Low_pressure_valves"."IN_valve_gate__ERROR_B"[8] OR
       "Low_pressure_valves"."IN_valve_gate__ERROR_B"[9]

   THEN
       "Low_pressure_valves".ERROR_IN_VALVE_ANY := TRUE;
   ELSE
       "Low_pressure_valves".ERROR_IN_VALVE_ANY := FALSE;
   END_IF;
END_REGION

REGION Network 5 (SCL): Неисправность любого шарового крана
   IF  NOT "SOVA_Modbus_Input".MB_Line[3, 1, 6] OR // Шаровой кран КР38.1 //
       NOT "SOVA_Modbus_Input".MB_Line[3, 2, 6] OR // Шаровой кран КР38.2 //
       NOT "SOVA_Modbus_Input".MB_Line[3, 3, 6] OR // Шаровой кран КР38.3 //
       NOT "SOVA_Modbus_Input".MB_Line[3, 4, 6] OR // Шаровой кран КР38.4 //
       NOT "SOVA_Modbus_Input".MB_Line[3, 5, 6] // Шаровой кран КР38.5 //
   THEN
       "Global".ERROR_BALL_VALVE_ANY := TRUE;
   ELSE
       "Global".ERROR_BALL_VALVE_ANY := FALSE;
   END_IF;
END_REGION

REGION Network 6: Неисправность основных магистральных кранов
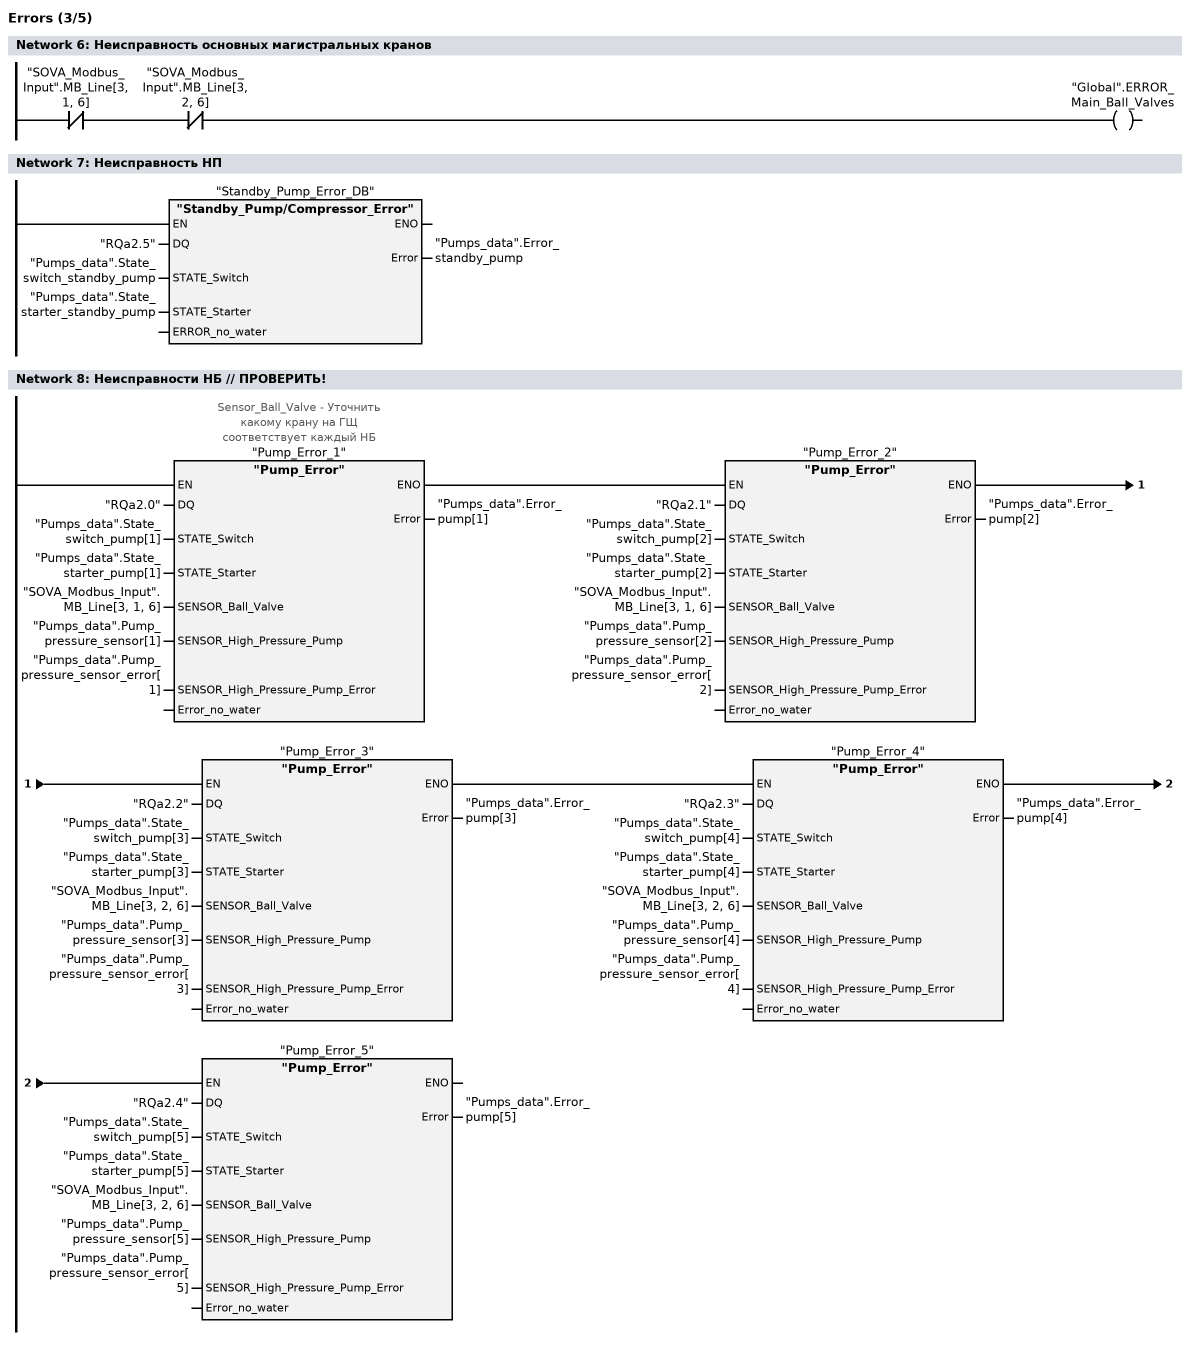
   RUNG wire#powerrail
      I_Contact( "SOVA_Modbus_Input".MB_Line[3, 1, 6] )
      I_Contact( "SOVA_Modbus_Input".MB_Line[3, 2, 6] )
      Coil( "Global".ERROR_Main_Ball_Valves )
   END_RUNG
   // the same network as SCL:
   "Global".ERROR_Main_Ball_Valves := NOT "SOVA_Modbus_Input".MB_Line[3, 1, 6] AND NOT "SOVA_Modbus_Input".MB_Line[3, 2, 6];
END_REGION

REGION Network 7: Неисправность НП
   RUNG wire#powerrail
      "Standby_Pump_Error_DB"(DQ := "RQa2.5", STATE_Switch := "Pumps_data".State_switch_standby_pump, STATE_Starter := "Pumps_data".State_starter_standby_pump, ERROR_no_water :=, Error => "Pumps_data".Error_standby_pump)
   END_RUNG
   // the same network as SCL:
   "Standby_Pump_Error_DB"(DQ := "RQa2.5",   // "Standby_Pump/Compressor_Error"
                           STATE_Switch := "Pumps_data".State_switch_standby_pump,
                           STATE_Starter := "Pumps_data".State_starter_standby_pump,
                           Error => "Pumps_data".Error_standby_pump);
END_REGION

REGION Network 8: Неисправности НБ // ПРОВЕРИТЬ!
   RUNG wire#powerrail
      "Pump_Error_1"(DQ := "RQa2.0", STATE_Switch := "Pumps_data".State_switch_pump[1], STATE_Starter := "Pumps_data".State_starter_pump[1], SENSOR_Ball_Valve := "SOVA_Modbus_Input".MB_Line[3, 1, 6], SENSOR_High_Pressure_Pump := "Pumps_data".Pump_pressure_sensor[1], SENSOR_High_Pressure_Pump_Error := "Pumps_data".Pump_pressure_sensor_error[1], Error_no_water :=, Error => "Pumps_data".Error_pump[1])   // Sensor_Ball_Valve - Уточнить какому крану на ГЩ соответствует каждый НБ
      "Pump_Error_2"(DQ := "RQa2.1", STATE_Switch := "Pumps_data".State_switch_pump[2], STATE_Starter := "Pumps_data".State_starter_pump[2], SENSOR_Ball_Valve := "SOVA_Modbus_Input".MB_Line[3, 1, 6], SENSOR_High_Pressure_Pump := "Pumps_data".Pump_pressure_sensor[2], SENSOR_High_Pressure_Pump_Error := "Pumps_data".Pump_pressure_sensor_error[2], Error_no_water :=, Error => "Pumps_data".Error_pump[2])
      "Pump_Error_3"(DQ := "RQa2.2", STATE_Switch := "Pumps_data".State_switch_pump[3], STATE_Starter := "Pumps_data".State_starter_pump[3], SENSOR_Ball_Valve := "SOVA_Modbus_Input".MB_Line[3, 2, 6], SENSOR_High_Pressure_Pump := "Pumps_data".Pump_pressure_sensor[3], SENSOR_High_Pressure_Pump_Error := "Pumps_data".Pump_pressure_sensor_error[3], Error_no_water :=, Error => "Pumps_data".Error_pump[3])
      "Pump_Error_4"(DQ := "RQa2.3", STATE_Switch := "Pumps_data".State_switch_pump[4], STATE_Starter := "Pumps_data".State_starter_pump[4], SENSOR_Ball_Valve := "SOVA_Modbus_Input".MB_Line[3, 2, 6], SENSOR_High_Pressure_Pump := "Pumps_data".Pump_pressure_sensor[4], SENSOR_High_Pressure_Pump_Error := "Pumps_data".Pump_pressure_sensor_error[4], Error_no_water :=, Error => "Pumps_data".Error_pump[4])
      "Pump_Error_5"(DQ := "RQa2.4", STATE_Switch := "Pumps_data".State_switch_pump[5], STATE_Starter := "Pumps_data".State_starter_pump[5], SENSOR_Ball_Valve := "SOVA_Modbus_Input".MB_Line[3, 2, 6], SENSOR_High_Pressure_Pump := "Pumps_data".Pump_pressure_sensor[5], SENSOR_High_Pressure_Pump_Error := "Pumps_data".Pump_pressure_sensor_error[5], Error_no_water :=, Error => "Pumps_data".Error_pump[5])
   END_RUNG
   // the same network as SCL:
   "Pump_Error_1"(DQ := "RQa2.0",   // "Pump_Error": Sensor_Ball_Valve - Уточнить какому крану на ГЩ соответствует каждый НБ
                  STATE_Switch := "Pumps_data".State_switch_pump[1],
                  STATE_Starter := "Pumps_data".State_starter_pump[1],
                  SENSOR_Ball_Valve := "SOVA_Modbus_Input".MB_Line[3, 1, 6],
                  SENSOR_High_Pressure_Pump := "Pumps_data".Pump_pressure_sensor[1],
                  SENSOR_High_Pressure_Pump_Error := "Pumps_data".Pump_pressure_sensor_error[1],
                  Error => "Pumps_data".Error_pump[1],
                  ENO => #_w1);
   "Pump_Error_2"(EN := #_w1,   // "Pump_Error"
                  DQ := "RQa2.1",
                  STATE_Switch := "Pumps_data".State_switch_pump[2],
                  STATE_Starter := "Pumps_data".State_starter_pump[2],
                  SENSOR_Ball_Valve := "SOVA_Modbus_Input".MB_Line[3, 1, 6],
                  SENSOR_High_Pressure_Pump := "Pumps_data".Pump_pressure_sensor[2],
                  SENSOR_High_Pressure_Pump_Error := "Pumps_data".Pump_pressure_sensor_error[2],
                  Error => "Pumps_data".Error_pump[2],
                  ENO => #_w2);
   "Pump_Error_3"(EN := #_w2,   // "Pump_Error"
                  DQ := "RQa2.2",
                  STATE_Switch := "Pumps_data".State_switch_pump[3],
                  STATE_Starter := "Pumps_data".State_starter_pump[3],
                  SENSOR_Ball_Valve := "SOVA_Modbus_Input".MB_Line[3, 2, 6],
                  SENSOR_High_Pressure_Pump := "Pumps_data".Pump_pressure_sensor[3],
                  SENSOR_High_Pressure_Pump_Error := "Pumps_data".Pump_pressure_sensor_error[3],
                  Error => "Pumps_data".Error_pump[3],
                  ENO => #_w3);
   "Pump_Error_4"(EN := #_w3,   // "Pump_Error"
                  DQ := "RQa2.3",
                  STATE_Switch := "Pumps_data".State_switch_pump[4],
                  STATE_Starter := "Pumps_data".State_starter_pump[4],
                  SENSOR_Ball_Valve := "SOVA_Modbus_Input".MB_Line[3, 2, 6],
                  SENSOR_High_Pressure_Pump := "Pumps_data".Pump_pressure_sensor[4],
                  SENSOR_High_Pressure_Pump_Error := "Pumps_data".Pump_pressure_sensor_error[4],
                  Error => "Pumps_data".Error_pump[4],
                  ENO => #_w4);
   IF #_w4 THEN
       "Pump_Error_5"(DQ := "RQa2.4",   // "Pump_Error"
                      STATE_Switch := "Pumps_data".State_switch_pump[5],
                      STATE_Starter := "Pumps_data".State_starter_pump[5],
                      SENSOR_Ball_Valve := "SOVA_Modbus_Input".MB_Line[3, 2, 6],
                      SENSOR_High_Pressure_Pump := "Pumps_data".Pump_pressure_sensor[5],
                      SENSOR_High_Pressure_Pump_Error := "Pumps_data".Pump_pressure_sensor_error[5],
                      Error => "Pumps_data".Error_pump[5]);
   END_IF;
END_REGION

REGION Network 9 (SCL): Неисправность всех насосов
   IF
       "Pumps_data".Error_pump[1] AND
       "Pumps_data".Error_pump[2] AND
       "Pumps_data".Error_pump[3] AND
       "Pumps_data".Error_pump[4] AND
       "Pumps_data".Error_pump[5]
   THEN
       "Pumps_data".ERROR_PUMPS_ALL := TRUE;
   ELSE
       "Pumps_data".ERROR_PUMPS_ALL := FALSE;
   END_IF;
END_REGION

REGION Network 10 (SCL): Неисправность любого насоса
   IF 
       "Pumps_data".Error_pump[1] OR
       "Pumps_data".Error_pump[2] OR
       "Pumps_data".Error_pump[3] OR
       "Pumps_data".Error_pump[4] OR
       "Pumps_data".Error_pump[5]
   THEN
       "Pumps_data".ERROR_PUMPS_ANY := TRUE;
   ELSE
       "Pumps_data".ERROR_PUMPS_ANY := FALSE;
   END_IF;
END_REGION

REGION Network 11: Неисправности УУС // ПРОВЕРИТЬ!
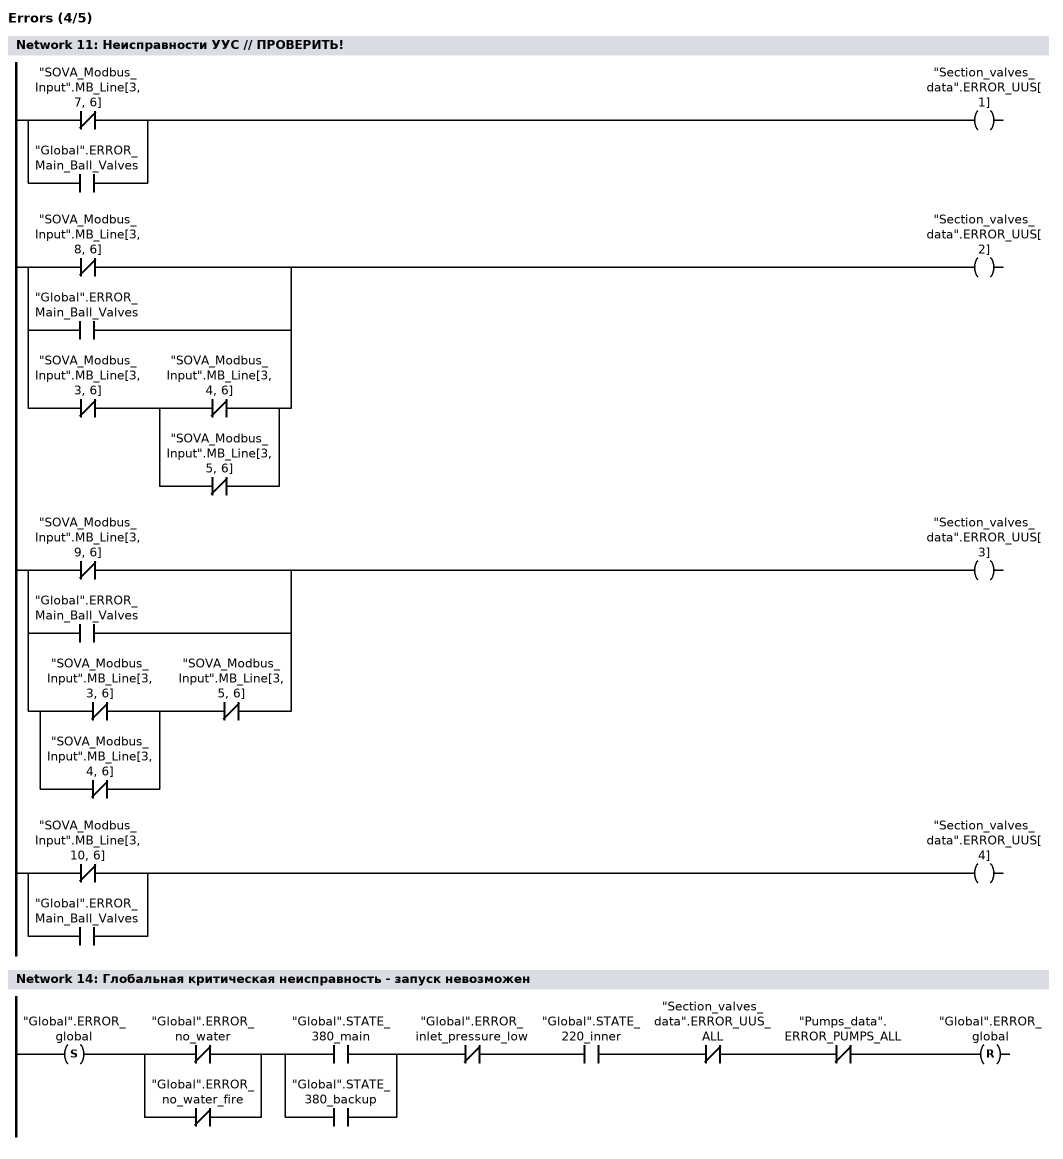
   RUNG wire#powerrail
      I_Contact( "SOVA_Modbus_Input".MB_Line[3, 7, 6] )
      wire#w1
      Coil( "Section_valves_data".ERROR_UUS[1] )
   END_RUNG
   RUNG wire#powerrail
      Contact( "Global".ERROR_Main_Ball_Valves )
   END_RUNG wire#w1
   RUNG wire#powerrail
      I_Contact( "SOVA_Modbus_Input".MB_Line[3, 8, 6] )
      wire#w2
      Coil( "Section_valves_data".ERROR_UUS[2] )
   END_RUNG
   RUNG wire#powerrail
      Contact( "Global".ERROR_Main_Ball_Valves )
   END_RUNG wire#w2
   RUNG wire#powerrail
      I_Contact( "SOVA_Modbus_Input".MB_Line[3, 3, 6] )
      wire#w3
      I_Contact( "SOVA_Modbus_Input".MB_Line[3, 4, 6] )
   END_RUNG wire#w2
   RUNG wire#w3
      I_Contact( "SOVA_Modbus_Input".MB_Line[3, 5, 6] )
   END_RUNG wire#w2
   RUNG wire#powerrail
      I_Contact( "SOVA_Modbus_Input".MB_Line[3, 9, 6] )
      wire#w4
      Coil( "Section_valves_data".ERROR_UUS[3] )
   END_RUNG
   RUNG wire#powerrail
      Contact( "Global".ERROR_Main_Ball_Valves )
   END_RUNG wire#w4
   RUNG wire#powerrail
      I_Contact( "SOVA_Modbus_Input".MB_Line[3, 3, 6] )
      wire#w5
      I_Contact( "SOVA_Modbus_Input".MB_Line[3, 5, 6] )
   END_RUNG wire#w4
   RUNG wire#powerrail
      I_Contact( "SOVA_Modbus_Input".MB_Line[3, 4, 6] )
   END_RUNG wire#w5
   RUNG wire#powerrail
      I_Contact( "SOVA_Modbus_Input".MB_Line[3, 10, 6] )
      wire#w6
      Coil( "Section_valves_data".ERROR_UUS[4] )
   END_RUNG
   RUNG wire#powerrail
      Contact( "Global".ERROR_Main_Ball_Valves )
   END_RUNG wire#w6
   // the same network as SCL:
   "Section_valves_data".ERROR_UUS[1] := NOT "SOVA_Modbus_Input".MB_Line[3, 7, 6] OR "Global".ERROR_Main_Ball_Valves;
   "Section_valves_data".ERROR_UUS[2] := NOT "SOVA_Modbus_Input".MB_Line[3, 8, 6] OR "Global".ERROR_Main_Ball_Valves OR (NOT "SOVA_Modbus_Input".MB_Line[3, 3, 6] AND (NOT "SOVA_Modbus_Input".MB_Line[3, 4, 6] OR NOT "SOVA_Modbus_Input".MB_Line[3, 5, 6]));
   "Section_valves_data".ERROR_UUS[3] := NOT "SOVA_Modbus_Input".MB_Line[3, 9, 6] OR "Global".ERROR_Main_Ball_Valves OR ((NOT "SOVA_Modbus_Input".MB_Line[3, 3, 6] OR NOT "SOVA_Modbus_Input".MB_Line[3, 4, 6]) AND NOT "SOVA_Modbus_Input".MB_Line[3, 5, 6]);
   "Section_valves_data".ERROR_UUS[4] := NOT "SOVA_Modbus_Input".MB_Line[3, 10, 6] OR "Global".ERROR_Main_Ball_Valves;
END_REGION

REGION Network 12 (SCL): Неисправность любого УУС
   IF "Section_valves_data".ERROR_UUS[1] OR // УУС.1 //
       "Section_valves_data".ERROR_UUS[2] OR // УУС.2 //
       "Section_valves_data".ERROR_UUS[3] OR // УУС.3 //
       "Section_valves_data".ERROR_UUS[4] // УУС.4 //
   THEN
       "Section_valves_data".ERROR_UUS_ANY := true;
   ELSE
       "Section_valves_data".ERROR_UUS_ANY := false;
   END_IF;
END_REGION

REGION Network 13 (SCL): Неисправность всех УУС
   IF "Section_valves_data".ERROR_UUS[1] AND // УУС.1 //
       "Section_valves_data".ERROR_UUS[2] AND // УУС.2 //
       "Section_valves_data".ERROR_UUS[3] AND // УУС.3 //
       "Section_valves_data".ERROR_UUS[4] // УУС.4 //
   THEN
       "Section_valves_data".ERROR_UUS_ALL := true;
   ELSE
       "Section_valves_data".ERROR_UUS_ALL := false;
   END_IF;
END_REGION

REGION Network 14: Глобальная критическая неисправность - запуск невозможен
   RUNG wire#powerrail
      S_Coil( "Global".ERROR_global )
      wire#w1
      I_Contact( "Global".ERROR_no_water )
      wire#w2
      Contact( "Global".STATE_380_main )
      wire#w3
      I_Contact( "Global".ERROR_inlet_pressure_low )
      Contact( "Global".STATE_220_inner )
      I_Contact( "Section_valves_data".ERROR_UUS_ALL )
      I_Contact( "Pumps_data".ERROR_PUMPS_ALL )
      R_Coil( "Global".ERROR_global )
   END_RUNG
   RUNG wire#w1
      I_Contact( "Global".ERROR_no_water_fire )
   END_RUNG wire#w2
   RUNG wire#w2
      Contact( "Global".STATE_380_backup )
   END_RUNG wire#w3
   // the same network as SCL:
   "Global".ERROR_global := TRUE;
   IF (NOT "Global".ERROR_no_water OR NOT "Global".ERROR_no_water_fire) AND ("Global".STATE_380_main OR "Global".STATE_380_backup) AND NOT "Global".ERROR_inlet_pressure_low AND "Global".STATE_220_inner AND NOT "Section_valves_data".ERROR_UUS_ALL AND NOT "Pumps_data".ERROR_PUMPS_ALL THEN
       "Global".ERROR_global := FALSE;
   END_IF;
END_REGION

REGION Network 15: Любая неисправность
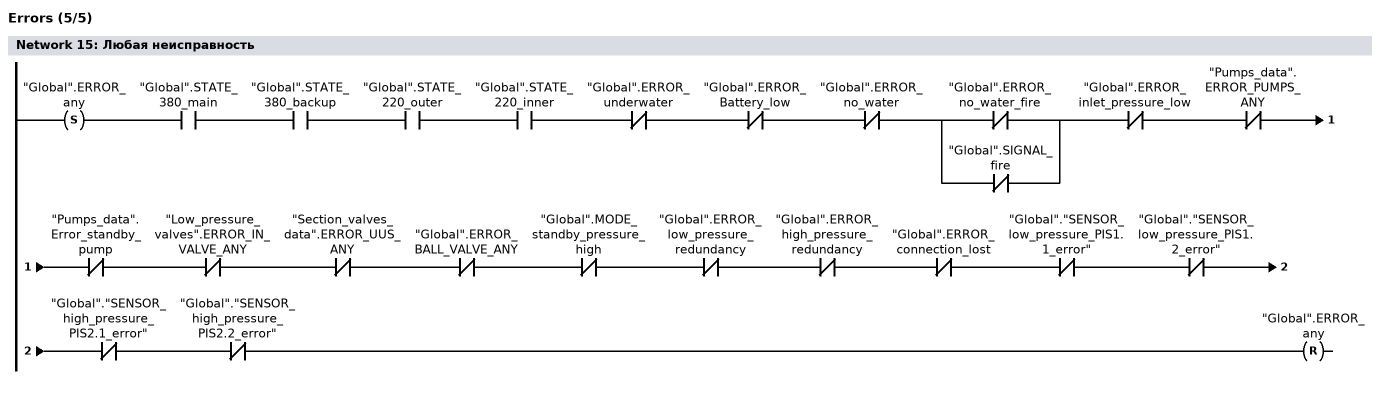
   RUNG wire#powerrail
      S_Coil( "Global".ERROR_any )
      Contact( "Global".STATE_380_main )
      Contact( "Global".STATE_380_backup )
      Contact( "Global".STATE_220_outer )
      Contact( "Global".STATE_220_inner )
      I_Contact( "Global".ERROR_underwater )
      I_Contact( "Global".ERROR_Battery_low )
      I_Contact( "Global".ERROR_no_water )
      wire#w1
      I_Contact( "Global".ERROR_no_water_fire )
      wire#w2
      I_Contact( "Global".ERROR_inlet_pressure_low )
      I_Contact( "Pumps_data".ERROR_PUMPS_ANY )
      I_Contact( "Pumps_data".Error_standby_pump )
      I_Contact( "Low_pressure_valves".ERROR_IN_VALVE_ANY )
      I_Contact( "Section_valves_data".ERROR_UUS_ANY )
      I_Contact( "Global".ERROR_BALL_VALVE_ANY )
      I_Contact( "Global".MODE_standby_pressure_high )
      I_Contact( "Global".ERROR_low_pressure_redundancy )
      I_Contact( "Global".ERROR_high_pressure_redundancy )
      I_Contact( "Global".ERROR_connection_lost )
      I_Contact( "Global"."SENSOR_low_pressure_PIS1.1_error" )
      I_Contact( "Global"."SENSOR_low_pressure_PIS1.2_error" )
      I_Contact( "Global"."SENSOR_high_pressure_PIS2.1_error" )
      I_Contact( "Global"."SENSOR_high_pressure_PIS2.2_error" )
      R_Coil( "Global".ERROR_any )
   END_RUNG
   RUNG wire#w1
      I_Contact( "Global".SIGNAL_fire )
   END_RUNG wire#w2
   // the same network as SCL:
   "Global".ERROR_any := TRUE;
   IF "Global".STATE_380_main AND "Global".STATE_380_backup AND "Global".STATE_220_outer AND "Global".STATE_220_inner AND NOT "Global".ERROR_underwater AND NOT "Global".ERROR_Battery_low AND NOT "Global".ERROR_no_water AND (NOT "Global".ERROR_no_water_fire OR NOT "Global".SIGNAL_fire) AND NOT "Global".ERROR_inlet_pressure_low AND NOT "Pumps_data".ERROR_PUMPS_ANY AND NOT "Pumps_data".Error_standby_pump AND NOT "Low_pressure_valves".ERROR_IN_VALVE_ANY AND NOT "Section_valves_data".ERROR_UUS_ANY AND NOT "Global".ERROR_BALL_VALVE_ANY AND NOT "Global".MODE_standby_pressure_high AND NOT "Global".ERROR_low_pressure_redundancy AND NOT "Global".ERROR_high_pressure_redundancy AND NOT "Global".ERROR_connection_lost AND NOT "Global"."SENSOR_low_pressure_PIS1.1_error" AND NOT "Global"."SENSOR_low_pressure_PIS1.2_error" AND NOT "Global"."SENSOR_high_pressure_PIS2.1_error" AND NOT "Global"."SENSOR_high_pressure_PIS2.2_error" THEN
       "Global".ERROR_any := FALSE;
   END_IF;
END_REGION
END_ORGANIZATION_BLOCK

ORGANIZATION_BLOCK "Buttons"   // OB124, LAD, ProgramCycle
TITLE = "Main Program Sweep (Cycle)"
{ S7_Optimized_Access := 'TRUE' }
VERSION : 0.1
   VAR_INPUT
      Initial_Call : Bool;   // Initial call of this OB
      Remanence : Bool;   // =True, if remanent data are available
   END_VAR
BEGIN

REGION Network 1: Звуковое оповещение и кнопка отключения звука
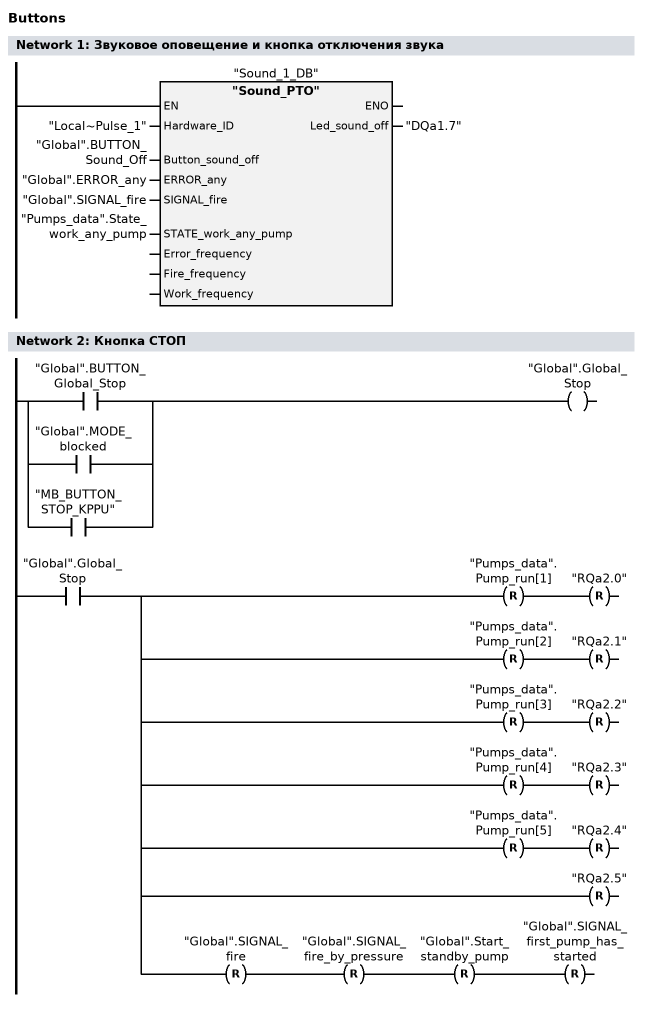
   RUNG wire#powerrail
      "Sound_1_DB"(Hardware_ID := "Local~Pulse_1", Button_sound_off := "Global".BUTTON_Sound_Off, ERROR_any := "Global".ERROR_any, SIGNAL_fire := "Global".SIGNAL_fire, STATE_work_any_pump := "Pumps_data".State_work_any_pump, Error_frequency :=, Fire_frequency :=, Work_frequency :=, Led_sound_off => "DQa1.7")
   END_RUNG
   // the same network as SCL:
   "Sound_1_DB"(Hardware_ID := "Local~Pulse_1",   // "Sound_PTO"
                Button_sound_off := "Global".BUTTON_Sound_Off,
                ERROR_any := "Global".ERROR_any,
                SIGNAL_fire := "Global".SIGNAL_fire,
                STATE_work_any_pump := "Pumps_data".State_work_any_pump,
                Led_sound_off => "DQa1.7");
END_REGION

REGION Network 2: Кнопка СТОП
   RUNG wire#powerrail
      Contact( "Global".BUTTON_Global_Stop )
      wire#w1
      Coil( "Global".Global_Stop )
   END_RUNG
   RUNG wire#powerrail
      Contact( "Global".MODE_blocked )
   END_RUNG wire#w1
   RUNG wire#powerrail
      Contact( "MB_BUTTON_STOP_KPPU" )
   END_RUNG wire#w1
   RUNG wire#powerrail
      Contact( "Global".Global_Stop )
      wire#w2
      R_Coil( "Pumps_data".Pump_run[1] )
      R_Coil( "RQa2.0" )
   END_RUNG
   RUNG wire#w2
      R_Coil( "Pumps_data".Pump_run[2] )
      R_Coil( "RQa2.1" )
   END_RUNG
   RUNG wire#w2
      R_Coil( "Pumps_data".Pump_run[3] )
      R_Coil( "RQa2.2" )
   END_RUNG
   RUNG wire#w2
      R_Coil( "Pumps_data".Pump_run[4] )
      R_Coil( "RQa2.3" )
   END_RUNG
   RUNG wire#w2
      R_Coil( "Pumps_data".Pump_run[5] )
      R_Coil( "RQa2.4" )
   END_RUNG
   RUNG wire#w2
      R_Coil( "RQa2.5" )
   END_RUNG
   RUNG wire#w2
      R_Coil( "Global".SIGNAL_fire )
      R_Coil( "Global".SIGNAL_fire_by_pressure )
      R_Coil( "Global".Start_standby_pump )
      R_Coil( "Global".SIGNAL_first_pump_has_started )
   END_RUNG
   // the same network as SCL:
   "Global".Global_Stop := "Global".BUTTON_Global_Stop OR "Global".MODE_blocked OR "MB_BUTTON_STOP_KPPU";
   IF "Global".Global_Stop THEN
       "Pumps_data".Pump_run[1] := FALSE;
       "RQa2.0" := FALSE;
       "Pumps_data".Pump_run[2] := FALSE;
       "RQa2.1" := FALSE;
       "Pumps_data".Pump_run[3] := FALSE;
       "RQa2.2" := FALSE;
       "Pumps_data".Pump_run[4] := FALSE;
       "RQa2.3" := FALSE;
       "Pumps_data".Pump_run[5] := FALSE;
       "RQa2.4" := FALSE;
       "RQa2.5" := FALSE;
       "Global".SIGNAL_fire := FALSE;
       "Global".SIGNAL_fire_by_pressure := FALSE;
       "Global".Start_standby_pump := FALSE;
       "Global".SIGNAL_first_pump_has_started := FALSE;
   END_IF;
END_REGION
END_ORGANIZATION_BLOCK

ORGANIZATION_BLOCK "Led"   // OB125, LAD, ProgramCycle
TITLE = "Main Program Sweep (Cycle)"
{ S7_Optimized_Access := 'TRUE' }
VERSION : 0.1
   VAR_INPUT
      Initial_Call : Bool;   // Initial call of this OB
      Remanence : Bool;   // =True, if remanent data are available
   END_VAR
   VAR_TEMP   // added for the SCL form of the ladder/FBD networks
      _w1 : Bool;
   END_VAR
BEGIN

REGION Network 1: Пожар, Пуск, Неисправность, Дежурный режим, Автоматика отклчена, Система отключена
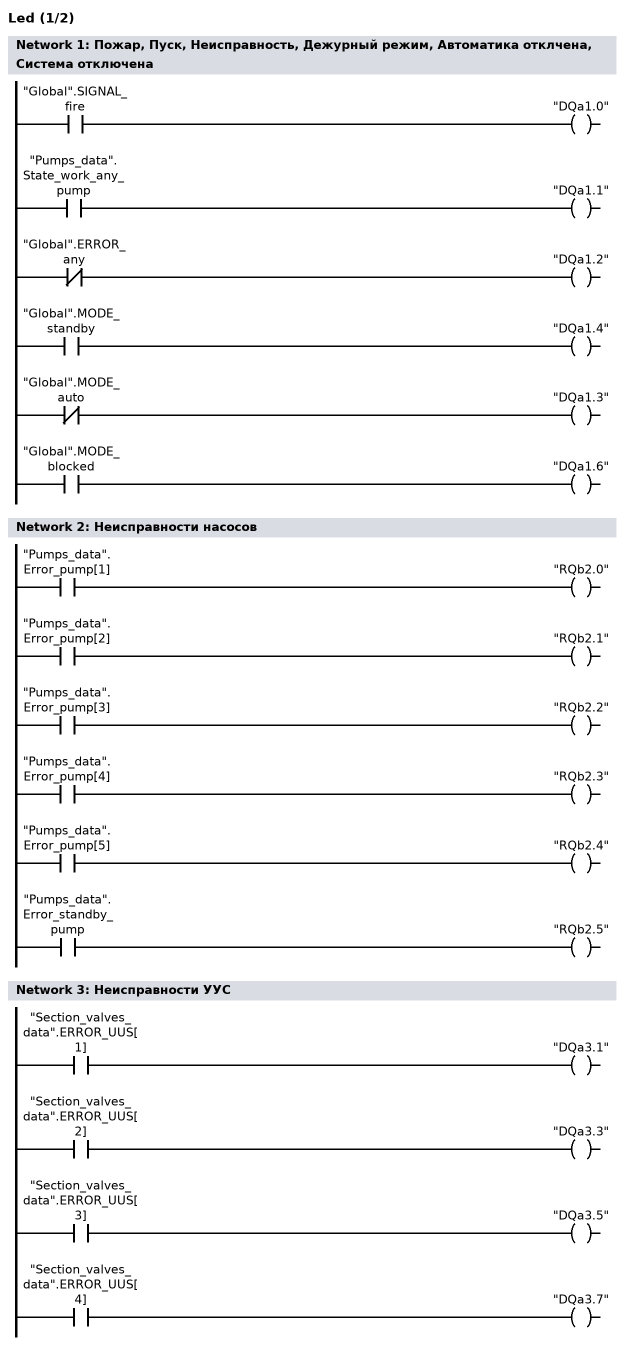
   RUNG wire#powerrail
      Contact( "Global".SIGNAL_fire )
      Coil( "DQa1.0" )
   END_RUNG
   RUNG wire#powerrail
      Contact( "Pumps_data".State_work_any_pump )
      Coil( "DQa1.1" )
   END_RUNG
   RUNG wire#powerrail
      I_Contact( "Global".ERROR_any )
      Coil( "DQa1.2" )
   END_RUNG
   RUNG wire#powerrail
      Contact( "Global".MODE_standby )
      Coil( "DQa1.4" )
   END_RUNG
   RUNG wire#powerrail
      I_Contact( "Global".MODE_auto )
      Coil( "DQa1.3" )
   END_RUNG
   RUNG wire#powerrail
      Contact( "Global".MODE_blocked )
      Coil( "DQa1.6" )
   END_RUNG
   // the same network as SCL:
   "DQa1.0" := "Global".SIGNAL_fire;
   "DQa1.1" := "Pumps_data".State_work_any_pump;
   "DQa1.2" := NOT "Global".ERROR_any;
   "DQa1.4" := "Global".MODE_standby;
   "DQa1.3" := NOT "Global".MODE_auto;
   "DQa1.6" := "Global".MODE_blocked;
END_REGION

REGION Network 2: Неисправности насосов
   RUNG wire#powerrail
      Contact( "Pumps_data".Error_pump[1] )
      Coil( "RQb2.0" )
   END_RUNG
   RUNG wire#powerrail
      Contact( "Pumps_data".Error_pump[2] )
      Coil( "RQb2.1" )
   END_RUNG
   RUNG wire#powerrail
      Contact( "Pumps_data".Error_pump[3] )
      Coil( "RQb2.2" )
   END_RUNG
   RUNG wire#powerrail
      Contact( "Pumps_data".Error_pump[4] )
      Coil( "RQb2.3" )
   END_RUNG
   RUNG wire#powerrail
      Contact( "Pumps_data".Error_pump[5] )
      Coil( "RQb2.4" )
   END_RUNG
   RUNG wire#powerrail
      Contact( "Pumps_data".Error_standby_pump )
      Coil( "RQb2.5" )
   END_RUNG
   // the same network as SCL:
   "RQb2.0" := "Pumps_data".Error_pump[1];
   "RQb2.1" := "Pumps_data".Error_pump[2];
   "RQb2.2" := "Pumps_data".Error_pump[3];
   "RQb2.3" := "Pumps_data".Error_pump[4];
   "RQb2.4" := "Pumps_data".Error_pump[5];
   "RQb2.5" := "Pumps_data".Error_standby_pump;
END_REGION

REGION Network 3: Неисправности УУС
   RUNG wire#powerrail
      Contact( "Section_valves_data".ERROR_UUS[1] )
      Coil( "DQa3.1" )
   END_RUNG
   RUNG wire#powerrail
      Contact( "Section_valves_data".ERROR_UUS[2] )
      Coil( "DQa3.3" )
   END_RUNG
   RUNG wire#powerrail
      Contact( "Section_valves_data".ERROR_UUS[3] )
      Coil( "DQa3.5" )
   END_RUNG
   RUNG wire#powerrail
      Contact( "Section_valves_data".ERROR_UUS[4] )
      Coil( "DQa3.7" )
   END_RUNG
   // the same network as SCL:
   "DQa3.1" := "Section_valves_data".ERROR_UUS[1];
   "DQa3.3" := "Section_valves_data".ERROR_UUS[2];
   "DQa3.5" := "Section_valves_data".ERROR_UUS[3];
   "DQa3.7" := "Section_valves_data".ERROR_UUS[4];
END_REGION

REGION Network 4: Срабатывание УУС
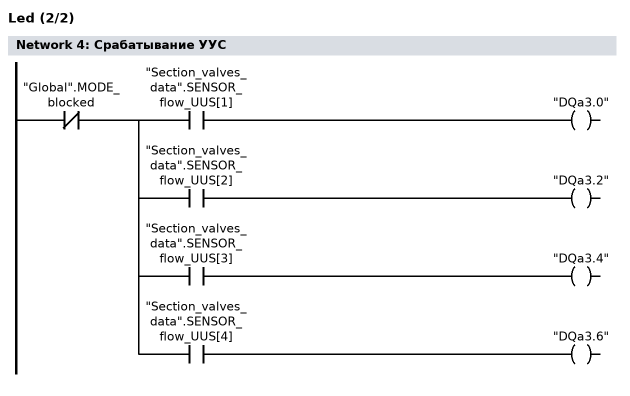
   RUNG wire#powerrail
      I_Contact( "Global".MODE_blocked )
      wire#w1
      Contact( "Section_valves_data".SENSOR_flow_UUS[1] )
      Coil( "DQa3.0" )
   END_RUNG
   RUNG wire#w1
      Contact( "Section_valves_data".SENSOR_flow_UUS[2] )
      Coil( "DQa3.2" )
   END_RUNG
   RUNG wire#w1
      Contact( "Section_valves_data".SENSOR_flow_UUS[3] )
      Coil( "DQa3.4" )
   END_RUNG
   RUNG wire#w1
      Contact( "Section_valves_data".SENSOR_flow_UUS[4] )
      Coil( "DQa3.6" )
   END_RUNG
   // the same network as SCL:
   #_w1 := NOT "Global".MODE_blocked;
   "DQa3.0" := #_w1 AND "Section_valves_data".SENSOR_flow_UUS[1];
   "DQa3.2" := #_w1 AND "Section_valves_data".SENSOR_flow_UUS[2];
   "DQa3.4" := #_w1 AND "Section_valves_data".SENSOR_flow_UUS[3];
   "DQa3.6" := #_w1 AND "Section_valves_data".SENSOR_flow_UUS[4];
END_REGION
END_ORGANIZATION_BLOCK

ORGANIZATION_BLOCK "Pumps"   // OB126, LAD, ProgramCycle
TITLE = "Main Program Sweep (Cycle)"
{ S7_Optimized_Access := 'TRUE' }
VERSION : 0.1
   VAR_INPUT
      Initial_Call : Bool;   // Initial call of this OB
      Remanence : Bool;   // =True, if remanent data are available
   END_VAR
   VAR_TEMP   // added for the SCL form of the ladder/FBD networks
      _w1 : Bool;
      _w2 : Bool;
   END_VAR
BEGIN

REGION Network 1: Работа жокей насоса
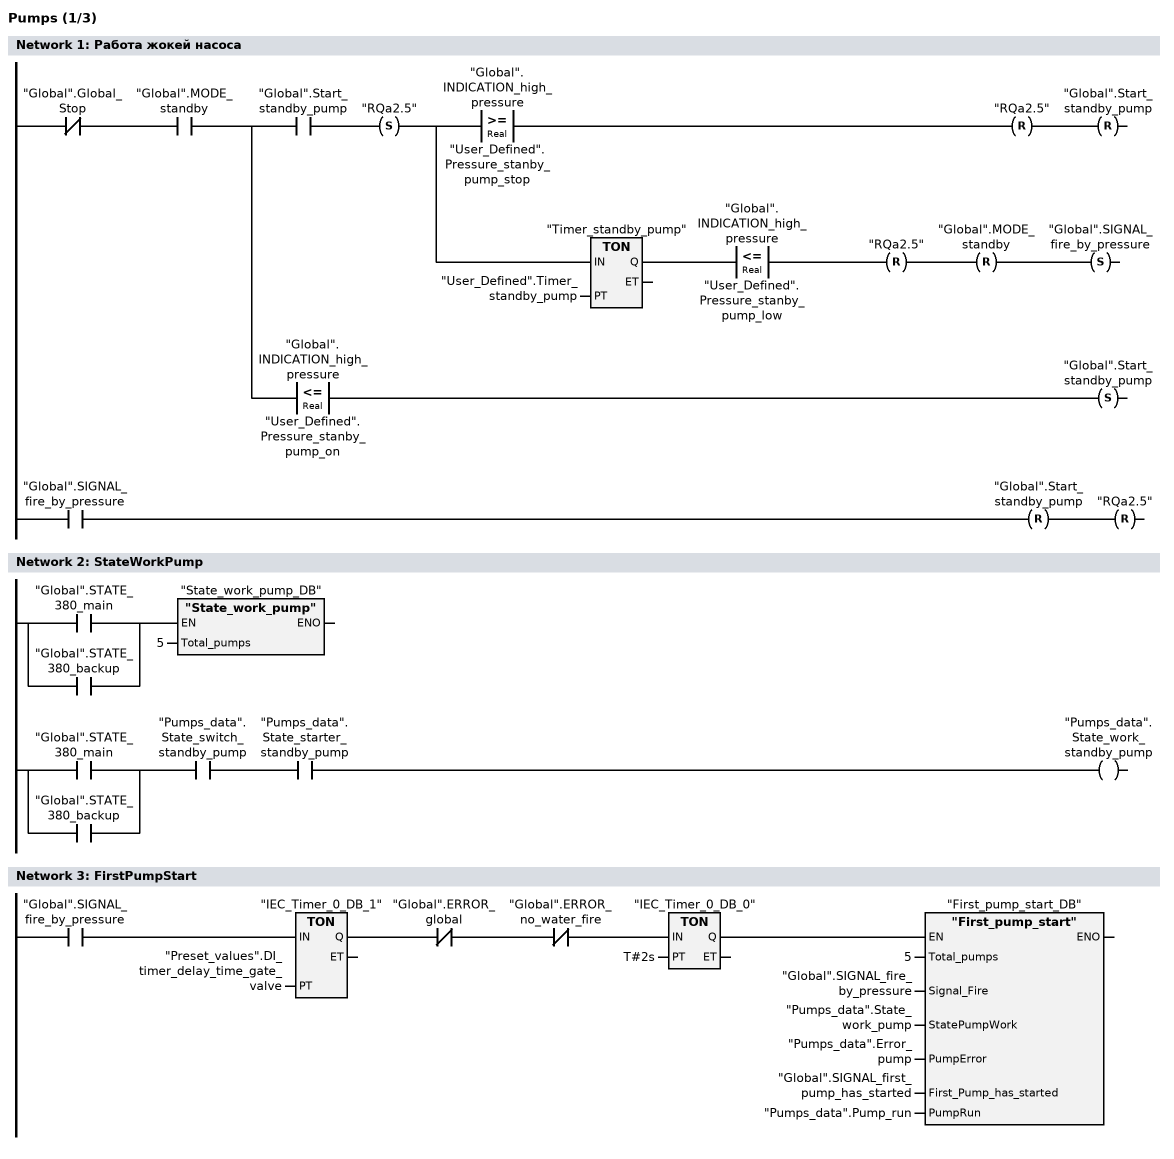
   #_w1 := NOT "Global".Global_Stop AND "Global".MODE_standby;
   #_w2 := #_w1 AND "Global".Start_standby_pump;
   IF #_w2 THEN "RQa2.5" := TRUE; END_IF;
   IF #_w2 AND ("Global".INDICATION_high_pressure >= "User_Defined".Pressure_stanby_pump_stop) THEN
       "RQa2.5" := FALSE;
       "Global".Start_standby_pump := FALSE;
   END_IF;
   "Timer_standby_pump".TON(IN := #_w2, PT := "User_Defined".Timer_standby_pump);
   IF "Timer_standby_pump".Q AND ("Global".INDICATION_high_pressure <= "User_Defined".Pressure_stanby_pump_low) THEN
       "RQa2.5" := FALSE;
       "Global".MODE_standby := FALSE;
       "Global".SIGNAL_fire_by_pressure := TRUE;
   END_IF;
   IF #_w1 AND ("Global".INDICATION_high_pressure <= "User_Defined".Pressure_stanby_pump_on) THEN
       "Global".Start_standby_pump := TRUE;
   END_IF;
   IF "Global".SIGNAL_fire_by_pressure THEN
       "Global".Start_standby_pump := FALSE;
       "RQa2.5" := FALSE;
   END_IF;
END_REGION

REGION Network 2: StateWorkPump
   RUNG wire#powerrail
      Contact( "Global".STATE_380_main )
      wire#w1
      "State_work_pump_DB"(Total_pumps := 5)
   END_RUNG
   RUNG wire#powerrail
      Contact( "Global".STATE_380_backup )
   END_RUNG wire#w1
   RUNG wire#powerrail
      Contact( "Global".STATE_380_main )
      wire#w2
      Contact( "Pumps_data".State_switch_standby_pump )
      Contact( "Pumps_data".State_starter_standby_pump )
      Coil( "Pumps_data".State_work_standby_pump )
   END_RUNG
   RUNG wire#powerrail
      Contact( "Global".STATE_380_backup )
   END_RUNG wire#w2
   // the same network as SCL:
   IF "Global".STATE_380_main OR "Global".STATE_380_backup THEN
       "State_work_pump_DB"(Total_pumps := 5);   // "State_work_pump"
   END_IF;
   "Pumps_data".State_work_standby_pump := ("Global".STATE_380_main OR "Global".STATE_380_backup) AND "Pumps_data".State_switch_standby_pump AND "Pumps_data".State_starter_standby_pump;
END_REGION

REGION Network 3: FirstPumpStart
   "IEC_Timer_0_DB_1".TON(IN := "Global".SIGNAL_fire_by_pressure,
                          PT := "Preset_values".DI_timer_delay_time_gate_valve);
   "IEC_Timer_0_DB_0".TON(IN := "IEC_Timer_0_DB_1".Q AND NOT "Global".ERROR_global AND NOT "Global".ERROR_no_water_fire,
                          PT := T#2s);
   IF "IEC_Timer_0_DB_0".Q THEN
       "First_pump_start_DB"(Total_pumps := 5,   // "First_pump_start"
                             Signal_Fire := "Global".SIGNAL_fire_by_pressure,
                             StatePumpWork := "Pumps_data".State_work_pump,
                             PumpError := "Pumps_data".Error_pump,
                             First_Pump_has_started := "Global".SIGNAL_first_pump_has_started,
                             PumpRun := "Pumps_data".Pump_run);
   END_IF;
END_REGION

REGION Network 4: Cascade
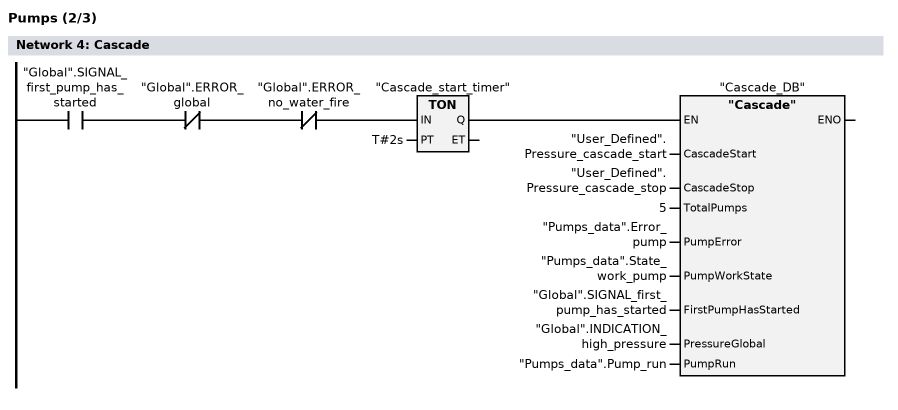
   "Cascade_start_timer".TON(IN := "Global".SIGNAL_first_pump_has_started AND NOT "Global".ERROR_global AND NOT "Global".ERROR_no_water_fire,
                           PT := T#2s);
   IF "Cascade_start_timer".Q THEN
       "Cascade_DB"(CascadeStart := "User_Defined".Pressure_cascade_start,   // "Cascade"
                    CascadeStop := "User_Defined".Pressure_cascade_stop,
                    TotalPumps := 5,
                    PumpError := "Pumps_data".Error_pump,
                    PumpWorkState := "Pumps_data".State_work_pump,
                    FirstPumpHasStarted := "Global".SIGNAL_first_pump_has_started,
                    PressureGlobal := "Global".INDICATION_high_pressure,
                    PumpRun := "Pumps_data".Pump_run);
   END_IF;
END_REGION

REGION Network 5: PumpRun
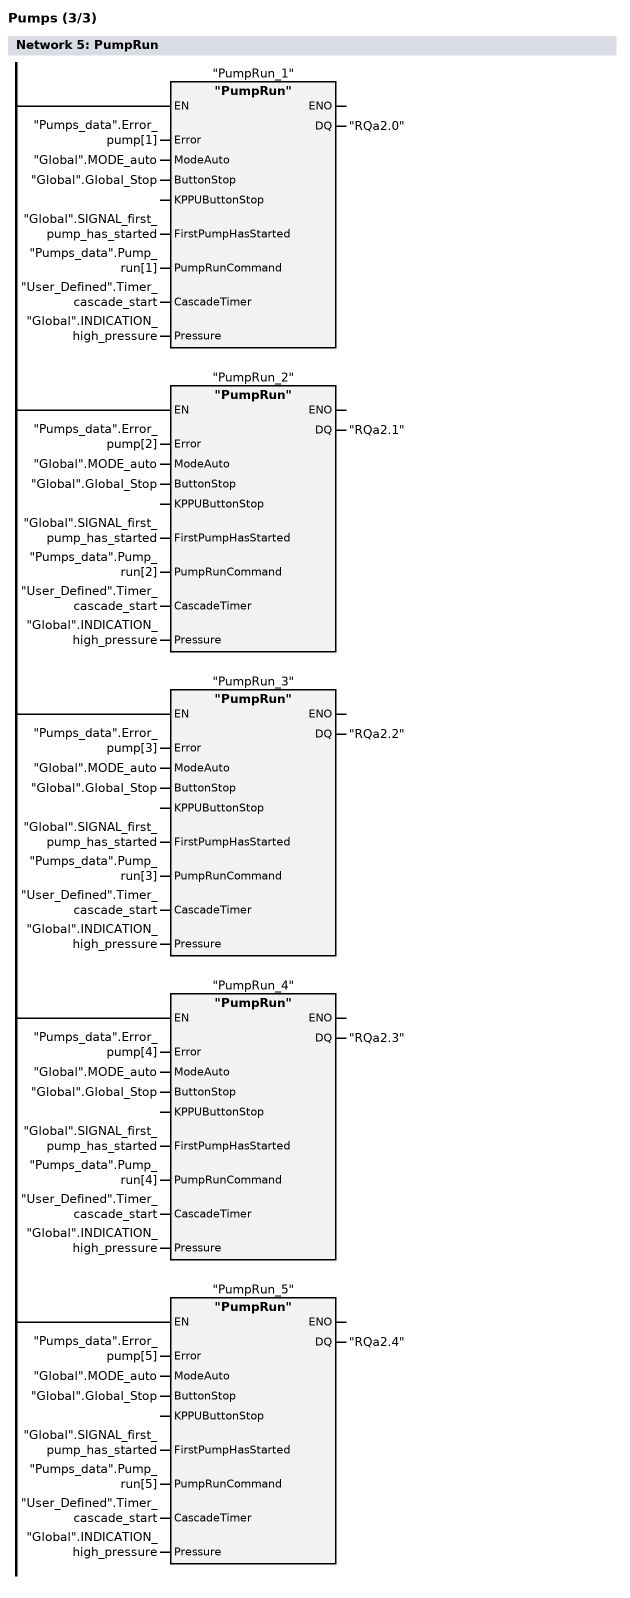
   RUNG wire#powerrail
      "PumpRun_1"(Error := "Pumps_data".Error_pump[1], ModeAuto := "Global".MODE_auto, ButtonStop := "Global".Global_Stop, KPPUButtonStop :=, FirstPumpHasStarted := "Global".SIGNAL_first_pump_has_started, PumpRunCommand := "Pumps_data".Pump_run[1], CascadeTimer := "User_Defined".Timer_cascade_start, Pressure := "Global".INDICATION_high_pressure, DQ => "RQa2.0")
   END_RUNG
   RUNG wire#powerrail
      "PumpRun_2"(Error := "Pumps_data".Error_pump[2], ModeAuto := "Global".MODE_auto, ButtonStop := "Global".Global_Stop, KPPUButtonStop :=, FirstPumpHasStarted := "Global".SIGNAL_first_pump_has_started, PumpRunCommand := "Pumps_data".Pump_run[2], CascadeTimer := "User_Defined".Timer_cascade_start, Pressure := "Global".INDICATION_high_pressure, DQ => "RQa2.1")
   END_RUNG
   RUNG wire#powerrail
      "PumpRun_3"(Error := "Pumps_data".Error_pump[3], ModeAuto := "Global".MODE_auto, ButtonStop := "Global".Global_Stop, KPPUButtonStop :=, FirstPumpHasStarted := "Global".SIGNAL_first_pump_has_started, PumpRunCommand := "Pumps_data".Pump_run[3], CascadeTimer := "User_Defined".Timer_cascade_start, Pressure := "Global".INDICATION_high_pressure, DQ => "RQa2.2")
   END_RUNG
   RUNG wire#powerrail
      "PumpRun_4"(Error := "Pumps_data".Error_pump[4], ModeAuto := "Global".MODE_auto, ButtonStop := "Global".Global_Stop, KPPUButtonStop :=, FirstPumpHasStarted := "Global".SIGNAL_first_pump_has_started, PumpRunCommand := "Pumps_data".Pump_run[4], CascadeTimer := "User_Defined".Timer_cascade_start, Pressure := "Global".INDICATION_high_pressure, DQ => "RQa2.3")
   END_RUNG
   RUNG wire#powerrail
      "PumpRun_5"(Error := "Pumps_data".Error_pump[5], ModeAuto := "Global".MODE_auto, ButtonStop := "Global".Global_Stop, KPPUButtonStop :=, FirstPumpHasStarted := "Global".SIGNAL_first_pump_has_started, PumpRunCommand := "Pumps_data".Pump_run[5], CascadeTimer := "User_Defined".Timer_cascade_start, Pressure := "Global".INDICATION_high_pressure, DQ => "RQa2.4")
   END_RUNG
   // the same network as SCL:
   "PumpRun_1"(Error := "Pumps_data".Error_pump[1],   // "PumpRun"
               ModeAuto := "Global".MODE_auto,
               ButtonStop := "Global".Global_Stop,
               FirstPumpHasStarted := "Global".SIGNAL_first_pump_has_started,
               PumpRunCommand := "Pumps_data".Pump_run[1],
               CascadeTimer := "User_Defined".Timer_cascade_start,
               Pressure := "Global".INDICATION_high_pressure,
               DQ => "RQa2.0");
   "PumpRun_2"(Error := "Pumps_data".Error_pump[2],   // "PumpRun"
               ModeAuto := "Global".MODE_auto,
               ButtonStop := "Global".Global_Stop,
               FirstPumpHasStarted := "Global".SIGNAL_first_pump_has_started,
               PumpRunCommand := "Pumps_data".Pump_run[2],
               CascadeTimer := "User_Defined".Timer_cascade_start,
               Pressure := "Global".INDICATION_high_pressure,
               DQ => "RQa2.1");
   "PumpRun_3"(Error := "Pumps_data".Error_pump[3],   // "PumpRun"
               ModeAuto := "Global".MODE_auto,
               ButtonStop := "Global".Global_Stop,
               FirstPumpHasStarted := "Global".SIGNAL_first_pump_has_started,
               PumpRunCommand := "Pumps_data".Pump_run[3],
               CascadeTimer := "User_Defined".Timer_cascade_start,
               Pressure := "Global".INDICATION_high_pressure,
               DQ => "RQa2.2");
   "PumpRun_4"(Error := "Pumps_data".Error_pump[4],   // "PumpRun"
               ModeAuto := "Global".MODE_auto,
               ButtonStop := "Global".Global_Stop,
               FirstPumpHasStarted := "Global".SIGNAL_first_pump_has_started,
               PumpRunCommand := "Pumps_data".Pump_run[4],
               CascadeTimer := "User_Defined".Timer_cascade_start,
               Pressure := "Global".INDICATION_high_pressure,
               DQ => "RQa2.3");
   "PumpRun_5"(Error := "Pumps_data".Error_pump[5],   // "PumpRun"
               ModeAuto := "Global".MODE_auto,
               ButtonStop := "Global".Global_Stop,
               FirstPumpHasStarted := "Global".SIGNAL_first_pump_has_started,
               PumpRunCommand := "Pumps_data".Pump_run[5],
               CascadeTimer := "User_Defined".Timer_cascade_start,
               Pressure := "Global".INDICATION_high_pressure,
               DQ => "RQa2.4");
END_REGION
END_ORGANIZATION_BLOCK

ORGANIZATION_BLOCK "Data_to_MB_HMI"   // OB127, LAD, ProgramCycle
TITLE = "Main Program Sweep (Cycle)"
{ S7_Optimized_Access := 'TRUE' }
VERSION : 0.1
   VAR_INPUT
      Initial_Call : Bool;   // Initial call of this OB
      Remanence : Bool;   // =True, if remanent data are available
   END_VAR
BEGIN

REGION Network 1 (SCL): Data to Modbus
   "MB_MODE_auto" := "Global".MODE_auto;
   "MB_MODE_manual" := "Global".MODE_manual;
   "MB_MODE_blocked" := "Global".MODE_blocked;
   "MB_MODE_standby" := "Global".MODE_standby;
   "MB_MODE_standby_pressure_high" := "Global".MODE_standby_pressure_high;
   "MB_BUTTON_Global_Stop" := "Global".BUTTON_Global_Stop;
   "MB_Global_Stop" := "Global".Global_Stop;
   "MB_BUTTON_Sound_Off" := "Global".BUTTON_Sound_Off;
   "MB_BUTTON_Led_Test" := "Global".BUTTON_Led_Test;
   "MB_STATE_380_main" := "Global".STATE_380_main;
   "MB_STATE_380_backup" := "Global".STATE_380_backup;
   "MB_STATE_220_inner" := "Global".STATE_220_inner;
   "MB_STATE_220_outer" := "Global".STATE_220_outer;
   "MB_STATE_door_opened" := "Global".STATE_door_opened;
   "MB_ERROR_underwater" := "Global".ERROR_underwater;
   "MB_ERROR_no_water" := "Global".ERROR_no_water;
   "MB_ERROR_no_water_fire" := "Global".ERROR_no_water_fire;
   "MB_ERROR_inlet_pressure_low" := "Global".ERROR_inlet_pressure_low;
   "MB_ERROR_global" := "Global".ERROR_global;
   "MB_ERROR_Main_Ball_Valves" := "Global".ERROR_Main_Ball_Valves;
   "MB_ERROR_BALL_VALVE_ANY" := "Global".ERROR_BALL_VALVE_ANY;
   "MB_ERROR_any" := "Global".ERROR_any;
   "MB_SIGNAL_fire" := "Global".SIGNAL_fire;
   "MB_SIGNAL_fire_by_pressure" := "Global".SIGNAL_fire_by_pressure;
   "MB_ERROR_high_pressure_redundancy" := "Global".ERROR_high_pressure_redundancy;
   "MB_ERROR_low_pressure_redundancy" := "Global".ERROR_low_pressure_redundancy;
   "MB_SIGNAL_first_pump_has_started" := "Global".SIGNAL_first_pump_has_started;
   "MB_Start_standby_pump" := "Global".Start_standby_pump;
   "MB_Secret_condition" := "Global".Secret_condition;
   "MB_ERROR_Battery_low" := "Global".ERROR_Battery_low;
   "MB_ERROR_connection_lost" := "Global".ERROR_connection_lost;
   "MB_ERROR_connection_lost_TOF" := "Global".ERROR_connection_lost_TOF;
   "MB_ERROR_connection_lost_TON" := "Global".ERROR_connection_lost_TON;
   "MB_SENSOR_low_pressure_PIS1.1_error" := "Global"."SENSOR_low_pressure_PIS1.1_error";
   "MB_SENSOR_low_pressure_PIS1.2_error" := "Global"."SENSOR_low_pressure_PIS1.2_error";
   "MB_SENSOR_high_pressure_PIS2.1_error" := "Global"."SENSOR_high_pressure_PIS2.1_error";
   "MB_SENSOR_high_pressure_PIS2.2_error" := "Global"."SENSOR_high_pressure_PIS2.2_error";
   "MB_IN_valve_gate__ERROR_B1" := "Low_pressure_valves"."IN_valve_gate__ERROR_B"[1];
   "MB_IN_valve_gate__ERROR_B2" := "Low_pressure_valves"."IN_valve_gate__ERROR_B"[2];
   "MB_IN_valve_gate__ERROR_B3" := "Low_pressure_valves"."IN_valve_gate__ERROR_B"[3];
   "MB_IN_valve_gate__ERROR_B4" := "Low_pressure_valves"."IN_valve_gate__ERROR_B"[4];
   "MB_IN_valve_gate__ERROR_B5" := "Low_pressure_valves"."IN_valve_gate__ERROR_B"[5];
   "MB_IN_valve_gate__ERROR_B6" := "Low_pressure_valves"."IN_valve_gate__ERROR_B"[6];
   "MB_IN_valve_gate__ERROR_B7" := "Low_pressure_valves"."IN_valve_gate__ERROR_B"[7];
   "MB_IN_valve_gate__ERROR_B8" := "Low_pressure_valves"."IN_valve_gate__ERROR_B"[8];
   "MB_IN_valve_gate__ERROR_B9" := "Low_pressure_valves"."IN_valve_gate__ERROR_B"[9];
   "MB_ERROR_IN_VALVE_ANY" := "Low_pressure_valves".ERROR_IN_VALVE_ANY;
   "MB_SENSOR_flow_UUS1" := "Section_valves_data".SENSOR_flow_UUS[1];
   "MB_SENSOR_flow_UUS2" := "Section_valves_data".SENSOR_flow_UUS[2];
   "MB_SENSOR_flow_UUS3" := "Section_valves_data".SENSOR_flow_UUS[3];
   "MB_SENSOR_flow_UUS4" := "Section_valves_data".SENSOR_flow_UUS[4];
   "MB_ERROR_UUS1" := "Section_valves_data".ERROR_UUS[1];
   "MB_ERROR_UUS2" := "Section_valves_data".ERROR_UUS[2];
   "MB_ERROR_UUS3" := "Section_valves_data".ERROR_UUS[3];
   "MB_ERROR_UUS4" := "Section_valves_data".ERROR_UUS[4];
   "MB_ERROR_UUS_ANY" := "Section_valves_data".ERROR_UUS_ANY;
   "MB_ERROR_UUS_ALL" := "Section_valves_data".ERROR_UUS_ALL;
   "MB_State_switch_pump1" := "Pumps_data".State_switch_pump[1];
   "MB_State_switch_pump2" := "Pumps_data".State_switch_pump[2];
   "MB_State_switch_pump3" := "Pumps_data".State_switch_pump[3];
   "MB_State_switch_pump4" := "Pumps_data".State_switch_pump[4];
   "MB_State_switch_pump5" := "Pumps_data".State_switch_pump[5];
   "MB_Error_pump1" := "Pumps_data".Error_pump[1];
   "MB_Error_pump2" := "Pumps_data".Error_pump[2];
   "MB_Error_pump3" := "Pumps_data".Error_pump[3];
   "MB_Error_pump4" := "Pumps_data".Error_pump[4];
   "MB_Error_pump5" := "Pumps_data".Error_pump[5];
   "MB_State_starter_pump1" := "Pumps_data".State_starter_pump[1];
   "MB_State_starter_pump2" := "Pumps_data".State_starter_pump[2];
   "MB_State_starter_pump3" := "Pumps_data".State_starter_pump[3];
   "MB_State_starter_pump4" := "Pumps_data".State_starter_pump[4];
   "MB_State_starter_pump5" := "Pumps_data".State_starter_pump[5];
   "MB_State_work_pump1" := "Pumps_data".State_work_pump[1];
   "MB_State_work_pump2" := "Pumps_data".State_work_pump[2];
   "MB_State_work_pump3" := "Pumps_data".State_work_pump[3];
   "MB_State_work_pump4" := "Pumps_data".State_work_pump[4];
   "MB_State_work_pump5" := "Pumps_data".State_work_pump[5];
   "MB_Pump_pressure_sensor_error1" := "Pumps_data".Pump_pressure_sensor_error[1];
   "MB_Pump_pressure_sensor_error2" := "Pumps_data".Pump_pressure_sensor_error[2];
   "MB_Pump_pressure_sensor_error3" := "Pumps_data".Pump_pressure_sensor_error[3];
   "MB_Pump_pressure_sensor_error4" := "Pumps_data".Pump_pressure_sensor_error[4];
   "MB_Pump_pressure_sensor_error5" := "Pumps_data".Pump_pressure_sensor_error[5];
   "MB_State_switch_standby_pump" := "Pumps_data".State_switch_standby_pump;
   "MB_Error_any_pump" := "Pumps_data".Error_any_pump;
   "MB_Error_standby_pump" := "Pumps_data".Error_standby_pump;
   "MB_State_starter_standby_pump" := "Pumps_data".State_starter_standby_pump;
   "MB_State_work_standby_pump" := "Pumps_data".State_work_standby_pump;
   "MB_State_work_any_pump" := "Pumps_data".State_work_any_pump;
   "MB_ERROR_PUMPS_ANY" := "Pumps_data".ERROR_PUMPS_ANY;
   "MB_ERROR_PUMPS_ALL" := "Pumps_data".ERROR_PUMPS_ALL;
   "MB_Low_pressure_valve_B1_open_OFF" := "SOVA_Modbus_Input".MB_Line[1, 1, 0];
   "MB_Low_pressure_valve_B1_open_NO_signal" := "SOVA_Modbus_Input".MB_Line[1, 1, 1];
   "MB_Low_pressure_valve_B1_open_short" := "SOVA_Modbus_Input".MB_Line[1, 1, 4];
   "MB_Low_pressure_valve_B1_open_brake" := "SOVA_Modbus_Input".MB_Line[1, 1, 5];
   "MB_Low_pressure_valve_B1_open_Signal" := "SOVA_Modbus_Input".MB_Line[1, 1, 6];
   "MB_Low_pressure_valve_B1_close_OFF" := "SOVA_Modbus_Input".MB_Line[1, 2, 0];
   "MB_Low_pressure_valve_B1_close_NO_signal" := "SOVA_Modbus_Input".MB_Line[1, 2, 1];
   "MB_Low_pressure_valve_B1_close_short" := "SOVA_Modbus_Input".MB_Line[1, 2, 4];
   "MB_Low_pressure_valve_B1_close_brake" := "SOVA_Modbus_Input".MB_Line[1, 2, 5];
   "MB_Low_pressure_valve_B1_close_Signal" := "SOVA_Modbus_Input".MB_Line[1, 2, 6];
   "MB_Low_pressure_valve_B2_open_OFF" := "SOVA_Modbus_Input".MB_Line[1, 3, 0];
   "MB_Low_pressure_valve_B2_open_NO_signal" := "SOVA_Modbus_Input".MB_Line[1, 3, 1];
   "MB_Low_pressure_valve_B2_open_short" := "SOVA_Modbus_Input".MB_Line[1, 3, 4];
   "MB_Low_pressure_valve_B2_open_brake" := "SOVA_Modbus_Input".MB_Line[1, 3, 5];
   "MB_Low_pressure_valve_B2_open_Signal" := "SOVA_Modbus_Input".MB_Line[1, 3, 6];
   "MB_Low_pressure_valve_B2_close_OFF" := "SOVA_Modbus_Input".MB_Line[1, 4, 0];
   "MB_Low_pressure_valve_B2_close_NO_signal" := "SOVA_Modbus_Input".MB_Line[1, 4, 1];
   "MB_Low_pressure_valve_B2_close_short" := "SOVA_Modbus_Input".MB_Line[1, 4, 4];
   "MB_Low_pressure_valve_B2_close_brake" := "SOVA_Modbus_Input".MB_Line[1, 4, 5];
   "MB_Low_pressure_valve_B2_close_Signal" := "SOVA_Modbus_Input".MB_Line[1, 4, 6];
   "MB_Low_pressure_valve_B3_open_OFF" := "SOVA_Modbus_Input".MB_Line[1, 5, 0];
   "MB_Low_pressure_valve_B3_open_NO_signal" := "SOVA_Modbus_Input".MB_Line[1, 5, 1];
   "MB_Low_pressure_valve_B3_open_short" := "SOVA_Modbus_Input".MB_Line[1, 5, 4];
   "MB_Low_pressure_valve_B3_open_brake" := "SOVA_Modbus_Input".MB_Line[1, 5, 5];
   "MB_Low_pressure_valve_B3_open_Signal" := "SOVA_Modbus_Input".MB_Line[1, 5, 6];
   "MB_Low_pressure_valve_B3_close_OFF" := "SOVA_Modbus_Input".MB_Line[1, 6, 0];
   "MB_Low_pressure_valve_B3_close_NO_signal" := "SOVA_Modbus_Input".MB_Line[1, 6, 1];
   "MB_Low_pressure_valve_B3_close_short" := "SOVA_Modbus_Input".MB_Line[1, 6, 4];
   "MB_Low_pressure_valve_B3_close_brake" := "SOVA_Modbus_Input".MB_Line[1, 6, 5];
   "MB_Low_pressure_valve_B3_close_Signal" := "SOVA_Modbus_Input".MB_Line[1, 6, 6];
   "MB_Low_pressure_valve_B4_open_OFF" := "SOVA_Modbus_Input".MB_Line[1, 7, 0];
   "MB_Low_pressure_valve_B4_open_NO_signal" := "SOVA_Modbus_Input".MB_Line[1, 7, 1];
   "MB_Low_pressure_valve_B4_open_short" := "SOVA_Modbus_Input".MB_Line[1, 7, 4];
   "MB_Low_pressure_valve_B4_open_brake" := "SOVA_Modbus_Input".MB_Line[1, 7, 5];
   "MB_Low_pressure_valve_B4_open_Signal" := "SOVA_Modbus_Input".MB_Line[1, 7, 6];
   "MB_Low_pressure_valve_B4_close_OFF" := "SOVA_Modbus_Input".MB_Line[1, 8, 0];
   "MB_Low_pressure_valve_B4_close_NO_signal" := "SOVA_Modbus_Input".MB_Line[1, 8, 1];
   "MB_Low_pressure_valve_B4_close_short" := "SOVA_Modbus_Input".MB_Line[1, 8, 4];
   "MB_Low_pressure_valve_B4_close_brake" := "SOVA_Modbus_Input".MB_Line[1, 8, 5];
   "MB_Low_pressure_valve_B4_close_Signal" := "SOVA_Modbus_Input".MB_Line[1, 8, 6];
   "MB_Low_pressure_valve_B5_open_OFF" := "SOVA_Modbus_Input".MB_Line[1, 9, 0];
   "MB_Low_pressure_valve_B5_open_NO_signal" := "SOVA_Modbus_Input".MB_Line[1, 9, 1];
   "MB_Low_pressure_valve_B5_open_short" := "SOVA_Modbus_Input".MB_Line[1, 9, 4];
   "MB_Low_pressure_valve_B5_open_brake" := "SOVA_Modbus_Input".MB_Line[1, 9, 5];
   "MB_Low_pressure_valve_B5_open_Signal" := "SOVA_Modbus_Input".MB_Line[1, 9, 6];
   "MB_Low_pressure_valve_B5_close_OFF" := "SOVA_Modbus_Input".MB_Line[1, 10, 0];
   "MB_Low_pressure_valve_B5_close_NO_signal" := "SOVA_Modbus_Input".MB_Line[1, 10, 1];
   "MB_Low_pressure_valve_B5_close_short" := "SOVA_Modbus_Input".MB_Line[1, 10, 4];
   "MB_Low_pressure_valve_B5_close_brake" := "SOVA_Modbus_Input".MB_Line[1, 10, 5];
   "MB_Low_pressure_valve_B5_close_Signal" := "SOVA_Modbus_Input".MB_Line[1, 10, 6];
   "MB_Low_pressure_valve_B6_open_OFF" := "SOVA_Modbus_Input".MB_Line[1, 11, 0];
   "MB_Low_pressure_valve_B6_open_NO_signal" := "SOVA_Modbus_Input".MB_Line[1, 11, 1];
   "MB_Low_pressure_valve_B6_open_short" := "SOVA_Modbus_Input".MB_Line[1, 11, 4];
   "MB_Low_pressure_valve_B6_open_brake" := "SOVA_Modbus_Input".MB_Line[1, 11, 5];
   "MB_Low_pressure_valve_B6_open_Signal" := "SOVA_Modbus_Input".MB_Line[1, 11, 6];
   "MB_Low_pressure_valve_B6_close_OFF" := "SOVA_Modbus_Input".MB_Line[1, 12, 0];
   "MB_Low_pressure_valve_B6_close_NO_signal" := "SOVA_Modbus_Input".MB_Line[1, 12, 1];
   "MB_Low_pressure_valve_B6_close_short" := "SOVA_Modbus_Input".MB_Line[1, 12, 4];
   "MB_Low_pressure_valve_B6_close_brake" := "SOVA_Modbus_Input".MB_Line[1, 12, 5];
   "MB_Low_pressure_valve_B6_close_Signal" := "SOVA_Modbus_Input".MB_Line[1, 12, 6];
   "MB_Low_pressure_valve_B7_open_OFF" := "SOVA_Modbus_Input".MB_Line[2, 1, 0];
   "MB_Low_pressure_valve_B7_open_NO_signal" := "SOVA_Modbus_Input".MB_Line[2, 1, 1];
   "MB_Low_pressure_valve_B7_open_short" := "SOVA_Modbus_Input".MB_Line[2, 1, 4];
   "MB_Low_pressure_valve_B7_open_brake" := "SOVA_Modbus_Input".MB_Line[2, 1, 5];
   "MB_Low_pressure_valve_B7_open_Signal" := "SOVA_Modbus_Input".MB_Line[2, 1, 6];
   "MB_Low_pressure_valve_B7_close_OFF" := "SOVA_Modbus_Input".MB_Line[2, 2, 0];
   "MB_Low_pressure_valve_B7_close_NO_signal" := "SOVA_Modbus_Input".MB_Line[2, 2, 1];
   "MB_Low_pressure_valve_B7_close_short" := "SOVA_Modbus_Input".MB_Line[2, 2, 4];
   "MB_Low_pressure_valve_B7_close_brake" := "SOVA_Modbus_Input".MB_Line[2, 2, 5];
   "MB_Low_pressure_valve_B7_close_Signal" := "SOVA_Modbus_Input".MB_Line[2, 2, 6];
   "MB_Low_pressure_valve_B8_open_OFF" := "SOVA_Modbus_Input".MB_Line[2, 3, 0];
   "MB_Low_pressure_valve_B8_open_NO_signal" := "SOVA_Modbus_Input".MB_Line[2, 3, 1];
   "MB_Low_pressure_valve_B8_open_short" := "SOVA_Modbus_Input".MB_Line[2, 3, 4];
   "MB_Low_pressure_valve_B8_open_brake" := "SOVA_Modbus_Input".MB_Line[2, 3, 5];
   "MB_Low_pressure_valve_B8_open_Signal" := "SOVA_Modbus_Input".MB_Line[2, 3, 6];
   "MB_Low_pressure_valve_B8_close_OFF" := "SOVA_Modbus_Input".MB_Line[2, 4, 0];
   "MB_Low_pressure_valve_B8_close_NO_signal" := "SOVA_Modbus_Input".MB_Line[2, 4, 1];
   "MB_Low_pressure_valve_B8_close_short" := "SOVA_Modbus_Input".MB_Line[2, 4, 4];
   "MB_Low_pressure_valve_B8_close_brake" := "SOVA_Modbus_Input".MB_Line[2, 4, 5];
   "MB_Low_pressure_valve_B8_close_Signal" := "SOVA_Modbus_Input".MB_Line[2, 4, 6];
   "MB_Low_pressure_valve_B9_open_OFF" := "SOVA_Modbus_Input".MB_Line[2, 5, 0];
   "MB_Low_pressure_valve_B9_open_NO_signal" := "SOVA_Modbus_Input".MB_Line[2, 5, 1];
   "MB_Low_pressure_valve_B9_open_short" := "SOVA_Modbus_Input".MB_Line[2, 5, 4];
   "MB_Low_pressure_valve_B9_open_brake" := "SOVA_Modbus_Input".MB_Line[2, 5, 5];
   "MB_Low_pressure_valve_B9_open_Signal" := "SOVA_Modbus_Input".MB_Line[2, 5, 6];
   "MB_Low_pressure_valve_B9_close_OFF" := "SOVA_Modbus_Input".MB_Line[2, 6, 0];
   "MB_Low_pressure_valve_B9_close_NO_signal" := "SOVA_Modbus_Input".MB_Line[2, 6, 1];
   "MB_Low_pressure_valve_B9_close_short" := "SOVA_Modbus_Input".MB_Line[2, 6, 4];
   "MB_Low_pressure_valve_B9_close_brake" := "SOVA_Modbus_Input".MB_Line[2, 6, 5];
   "MB_Low_pressure_valve_B9_close_Signal" := "SOVA_Modbus_Input".MB_Line[2, 6, 6];
   "MB_Ball_valve_K38.1_open_OFF" := "SOVA_Modbus_Input".MB_Line[3, 1, 0];
   "MB_Ball_valve_K38.1_open_NO_signal" := "SOVA_Modbus_Input".MB_Line[3, 1, 1];
   "MB_Ball_valve_K38.1_open_short" := "SOVA_Modbus_Input".MB_Line[3, 1, 4];
   "MB_Ball_valve_K38.1_open_brake" := "SOVA_Modbus_Input".MB_Line[3, 1, 5];
   "MB_Ball_valve_K38.1_open_Signal" := "SOVA_Modbus_Input".MB_Line[3, 1, 6];
   "MB_Ball_valve_K38.2_open_OFF" := "SOVA_Modbus_Input".MB_Line[3, 2, 0];
   "MB_Ball_valve_K38.2_open_NO_signal" := "SOVA_Modbus_Input".MB_Line[3, 2, 1];
   "MB_Ball_valve_K38.2_open_short" := "SOVA_Modbus_Input".MB_Line[3, 2, 4];
   "MB_Ball_valve_K38.2_open_brake" := "SOVA_Modbus_Input".MB_Line[3, 2, 5];
   "MB_Ball_valve_K38.2_open_Signal" := "SOVA_Modbus_Input".MB_Line[3, 2, 6];
   "MB_Ball_valve_K38.3_open_OFF" := "SOVA_Modbus_Input".MB_Line[3, 3, 0];
   "MB_Ball_valve_K38.3_open_NO_signal" := "SOVA_Modbus_Input".MB_Line[3, 3, 1];
   "MB_Ball_valve_K38.3_open_short" := "SOVA_Modbus_Input".MB_Line[3, 3, 4];
   "MB_Ball_valve_K38.3_open_brake" := "SOVA_Modbus_Input".MB_Line[3, 3, 5];
   "MB_Ball_valve_K38.3_open_Signal" := "SOVA_Modbus_Input".MB_Line[3, 3, 6];
   "MB_Ball_valve_K38.4_open_OFF" := "SOVA_Modbus_Input".MB_Line[3, 4, 0];
   "MB_Ball_valve_K38.4_open_NO_signal" := "SOVA_Modbus_Input".MB_Line[3, 4, 1];
   "MB_Ball_valve_K38.4_open_short" := "SOVA_Modbus_Input".MB_Line[3, 4, 4];
   "MB_Ball_valve_K38.4_open_brake" := "SOVA_Modbus_Input".MB_Line[3, 4, 5];
   "MB_Ball_valve_K38.4_open_Signal" := "SOVA_Modbus_Input".MB_Line[3, 4, 6];
   "MB_Ball_valve_K38.5_open_OFF" := "SOVA_Modbus_Input".MB_Line[3, 5, 0];
   "MB_Ball_valve_K38.5_open_NO_signal" := "SOVA_Modbus_Input".MB_Line[3, 5, 1];
   "MB_Ball_valve_K38.5_open_short" := "SOVA_Modbus_Input".MB_Line[3, 5, 4];
   "MB_Ball_valve_K38.5_open_brake" := "SOVA_Modbus_Input".MB_Line[3, 5, 5];
   "MB_Ball_valve_K38.5_open_Signal" := "SOVA_Modbus_Input".MB_Line[3, 5, 6];
   "MB_UUS.1_open_OFF" := "SOVA_Modbus_Input".MB_Line[3, 7, 0];
   "MB_UUS.1_open_NO_signal" := "SOVA_Modbus_Input".MB_Line[3, 7, 1];
   "MB_UUS.1_open_short" := "SOVA_Modbus_Input".MB_Line[3, 7, 4];
   "MB_UUS.1_open_brake" := "SOVA_Modbus_Input".MB_Line[3, 7, 5];
   "MB_UUS.1_open_Signal" := "SOVA_Modbus_Input".MB_Line[3, 7, 6];
   "MB_UUS.2_open_OFF" := "SOVA_Modbus_Input".MB_Line[3, 8, 0];
   "MB_UUS.2_open_NO_signal" := "SOVA_Modbus_Input".MB_Line[3, 8, 1];
   "MB_UUS.2_open_short" := "SOVA_Modbus_Input".MB_Line[3, 8, 4];
   "MB_UUS.2_open_brake" := "SOVA_Modbus_Input".MB_Line[3, 8, 5];
   "MB_UUS.2_open_Signal" := "SOVA_Modbus_Input".MB_Line[3, 8, 6];
   "MB_UUS.3_open_OFF" := "SOVA_Modbus_Input".MB_Line[3, 9, 0];
   "MB_UUS.3_open_NO_signal" := "SOVA_Modbus_Input".MB_Line[3, 9, 1];
   "MB_UUS.3_open_short" := "SOVA_Modbus_Input".MB_Line[3, 9, 4];
   "MB_UUS.3_open_brake" := "SOVA_Modbus_Input".MB_Line[3, 9, 5];
   "MB_UUS.3_open_Signal" := "SOVA_Modbus_Input".MB_Line[3, 9, 6];
   "MB_UUS.4_open_OFF" := "SOVA_Modbus_Input".MB_Line[3, 10, 0];
   "MB_UUS.4_open_NO_signal" := "SOVA_Modbus_Input".MB_Line[3, 10, 1];
   "MB_UUS.4_open_short" := "SOVA_Modbus_Input".MB_Line[3, 10, 4];
   "MB_UUS.4_open_brake" := "SOVA_Modbus_Input".MB_Line[3, 10, 5];
   "MB_UUS.4_open_Signal" := "SOVA_Modbus_Input".MB_Line[3, 10, 6];
   "MB_SENSOR_low_pressure_PIS1.1" := "Global"."SENSOR_low_pressure_PIS1.1";
   "MB_SENSOR_low_pressure_PIS1.2" := "Global"."SENSOR_low_pressure_PIS1.2";
   "MB_SENSOR_high_pressure_PIS2.1" := "Global"."SENSOR_high_pressure_PIS2.1";
   "MB_SENSOR_high_pressure_PIS2.2" := "Global"."SENSOR_high_pressure_PIS2.2";
   "MB_INDICATION_high_pressure" := "Global".INDICATION_high_pressure;
   "MB_INDICATION_low_pressure" := "Global".INDICATION_low_pressure;
   "MB_Pump_pressure_sensor1" := "Pumps_data".Pump_pressure_sensor[1];
   "MB_Pump_pressure_sensor2" := "Pumps_data".Pump_pressure_sensor[2];
   "MB_Pump_pressure_sensor3" := "Pumps_data".Pump_pressure_sensor[3];
   "MB_Pump_pressure_sensor4" := "Pumps_data".Pump_pressure_sensor[4];
   "MB_Pump_pressure_sensor5" := "Pumps_data".Pump_pressure_sensor[5];
END_REGION

